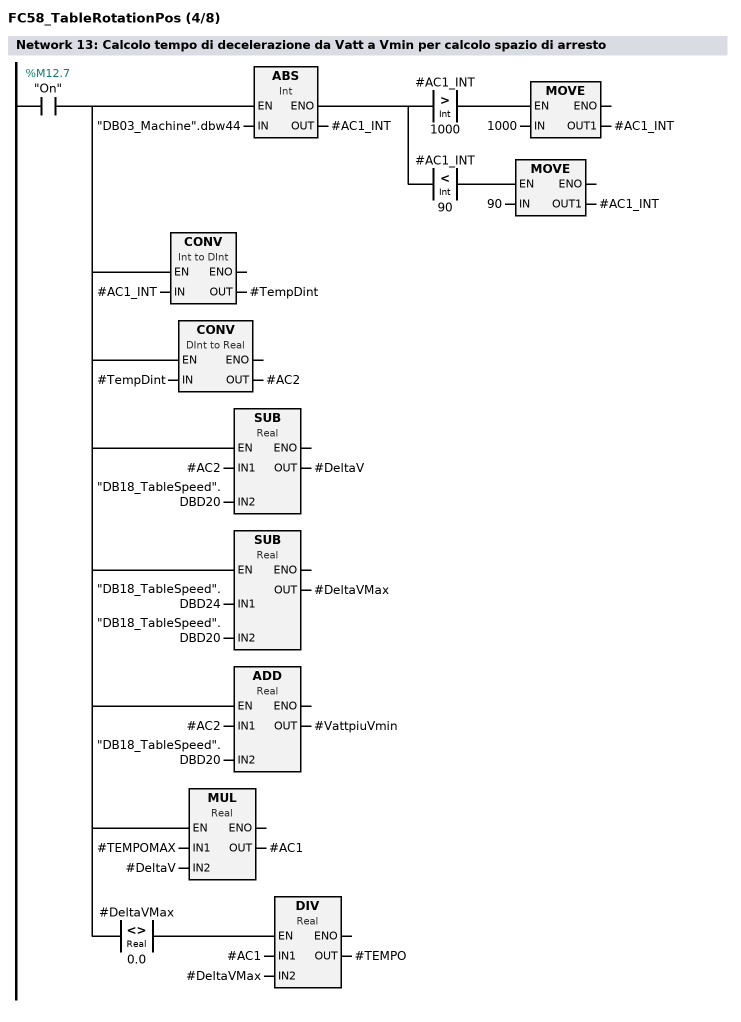
   RUNG wire#powerrail
      Contact( "On" )
      wire#w1
      { S7_Templates := "SrcType := Int" } Abs(in := "DB03_Machine".dbw44, out => #AC1_INT)
      wire#w2
      { S7_Templates := "SrcType := Int" } GT_Contact(in1 := #AC1_INT, in2 := 1000)
      Move(in := 1000, out1 => #AC1_INT)
   END_RUNG
   RUNG wire#w2
      { S7_Templates := "SrcType := Int" } LT_Contact(in1 := #AC1_INT, in2 := 90)
      Move(in := 90, out1 => #AC1_INT)
   END_RUNG
   RUNG wire#w1
      { S7_Templates := "[SrcType := Int, DestType := DInt]"; S7_GenerateENO := "TRUE" } Convert(in := #AC1_INT, out => #TempDint)
   END_RUNG
   RUNG wire#w1
      { S7_Templates := "[SrcType := DInt, DestType := Real]"; S7_GenerateENO := "TRUE" } Convert(in := #TempDint, out => #AC2)
   END_RUNG
   RUNG wire#w1
      { S7_Templates := "SrcType := Real"; S7_GenerateENO := "TRUE" } Sub(in1 := #AC2, in2 := "DB18_TableSpeed".DBD20, out => #DeltaV)
   END_RUNG
   RUNG wire#w1
      { S7_Templates := "SrcType := Real"; S7_GenerateENO := "TRUE" } Sub(in1 := "DB18_TableSpeed".DBD24, in2 := "DB18_TableSpeed".DBD20, out => #DeltaVMax)
   END_RUNG
   RUNG wire#w1
      { S7_Templates := "SrcType := Real"; S7_GenerateENO := "TRUE" } Add(in1 := #AC2, in2 := "DB18_TableSpeed".DBD20, out => #VattpiuVmin)
   END_RUNG
   RUNG wire#w1
      { S7_Templates := "SrcType := Real"; S7_GenerateENO := "TRUE" } Mul(in1 := #TEMPOMAX, in2 := #DeltaV, out => #AC1)
   END_RUNG
   RUNG wire#w1
      { S7_Templates := "SrcType := Real" } NE_Contact(in1 := #DeltaVMax, in2 := 0.0)
      { S7_Templates := "SrcType := Real"; S7_GenerateENO := "TRUE" } Div(in1 := #AC1, in2 := #DeltaVMax, out => #TEMPO)
   END_RUNG
   // the same network as SCL:
   IF "On" THEN #AC1_INT := ABS("DB03_Machine".dbw44); END_IF;
   IF "On" AND (#AC1_INT > 1000) THEN #AC1_INT := 1000; END_IF;
   IF "On" AND (#AC1_INT < 90) THEN #AC1_INT := 90; END_IF;
   IF "On" THEN
       #TempDint := INT_TO_DINT(#AC1_INT);
       #AC2 := DINT_TO_REAL(#TempDint);
       #DeltaV := #AC2 - "DB18_TableSpeed".DBD20;
       #DeltaVMax := "DB18_TableSpeed".DBD24 - "DB18_TableSpeed".DBD20;
       #VattpiuVmin := #AC2 + "DB18_TableSpeed".DBD20;
       #AC1 := #TEMPOMAX * #DeltaV;
   END_IF;
   IF "On" AND (#DeltaVMax <> 0.0) THEN #TEMPO := #AC1 / #DeltaVMax; END_IF;
END_REGION

REGION Network 14: Decelerazione
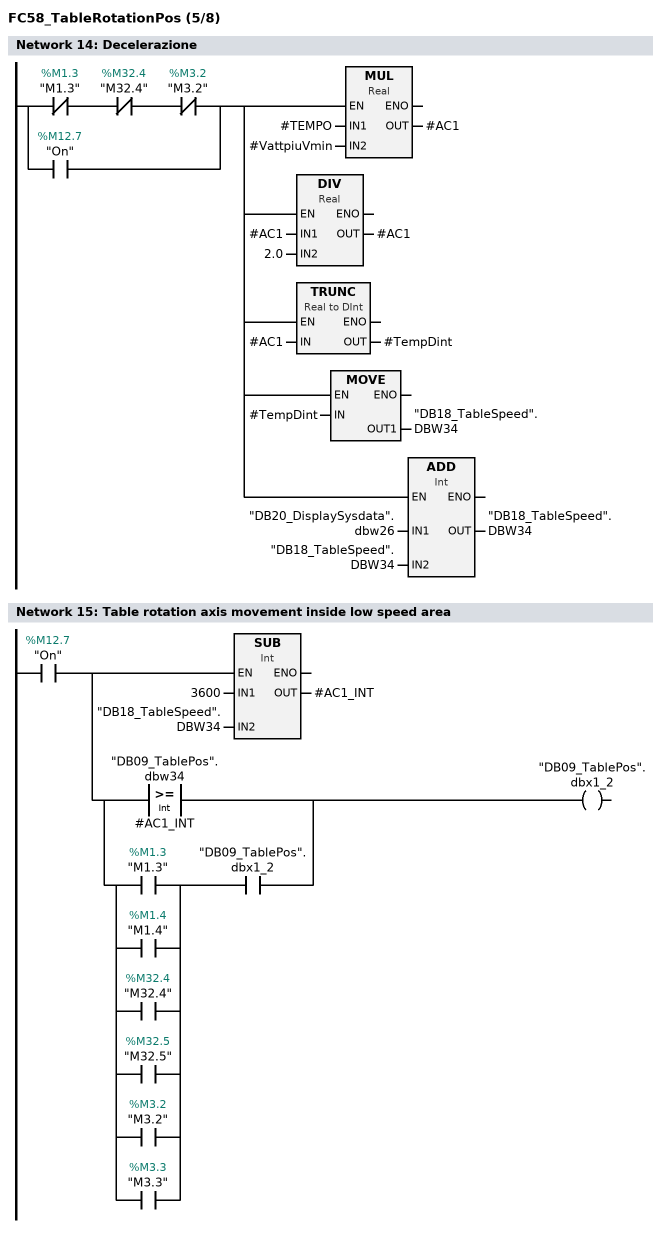
   RUNG wire#powerrail
      I_Contact( "M1.3" )
      I_Contact( "M32.4" )
      I_Contact( "M3.2" )
      wire#w1
      { S7_Templates := "SrcType := Real"; S7_GenerateENO := "TRUE" } Mul(in1 := #TEMPO, in2 := #VattpiuVmin, out => #AC1)
   END_RUNG
   RUNG wire#powerrail
      Contact( "On" )
   END_RUNG wire#w1
   RUNG wire#w1
      { S7_Templates := "SrcType := Real"; S7_GenerateENO := "TRUE" } Div(in1 := #AC1, in2 := 2.0, out => #AC1)
   END_RUNG
   RUNG wire#w1
      { S7_Templates := "[SrcType := Real, DestType := DInt]"; S7_GenerateENO := "TRUE" } Trunc(in := #AC1, out => #TempDint)
   END_RUNG
   RUNG wire#w1
      { S7_GenerateENO := "TRUE" } Move(in := #TempDint, out1 => "DB18_TableSpeed".DBW34)
   END_RUNG
   RUNG wire#w1
      { S7_Templates := "SrcType := Int"; S7_GenerateENO := "TRUE" } Add(in1 := "DB20_DisplaySysdata".dbw26, in2 := "DB18_TableSpeed".DBW34, out => "DB18_TableSpeed".DBW34)
   END_RUNG
   // the same network as SCL:
   IF (NOT "M1.3" AND NOT "M32.4" AND NOT "M3.2") OR "On" THEN
       #AC1 := #TEMPO * #VattpiuVmin;
       #AC1 := #AC1 / 2.0;
       #TempDint := TRUNC(#AC1);
       "DB18_TableSpeed".DBW34 := #TempDint;
       "DB18_TableSpeed".DBW34 := "DB20_DisplaySysdata".dbw26 + "DB18_TableSpeed".DBW34;
   END_IF;
END_REGION

REGION Network 15: Table rotation axis movement inside low speed area
   RUNG wire#powerrail
      Contact( "On" )
      wire#w1
      { S7_Templates := "SrcType := Int"; S7_GenerateENO := "TRUE" } Sub(in1 := 3600, in2 := "DB18_TableSpeed".DBW34, out => #AC1_INT)
   END_RUNG
   RUNG wire#w1
      { S7_Templates := "SrcType := Int" } GE_Contact(in1 := "DB09_TablePos".dbw34, in2 := #AC1_INT)
      wire#w2
      Coil( "DB09_TablePos".dbx1_2 )
   END_RUNG
   RUNG wire#w1
      Contact( "M1.3" )
      wire#w3
      Contact( "DB09_TablePos".dbx1_2 )
   END_RUNG wire#w2
   RUNG wire#w1
      Contact( "M1.4" )
   END_RUNG wire#w3
   RUNG wire#w1
      Contact( "M32.4" )
   END_RUNG wire#w3
   RUNG wire#w1
      Contact( "M32.5" )
   END_RUNG wire#w3
   RUNG wire#w1
      Contact( "M3.2" )
   END_RUNG wire#w3
   RUNG wire#w1
      Contact( "M3.3" )
   END_RUNG wire#w3
   // the same network as SCL:
   IF "On" THEN #AC1_INT := 3600 - "DB18_TableSpeed".DBW34; END_IF;
   "DB09_TablePos".dbx1_2 := "On" AND (("DB09_TablePos".dbw34 >= #AC1_INT) OR (("M1.3" OR "M1.4" OR "M32.4" OR "M32.5" OR "M3.2" OR "M3.3") AND "DB09_TablePos".dbx1_2));
END_REGION

REGION Network 16: Table rotation position loading/Unloading
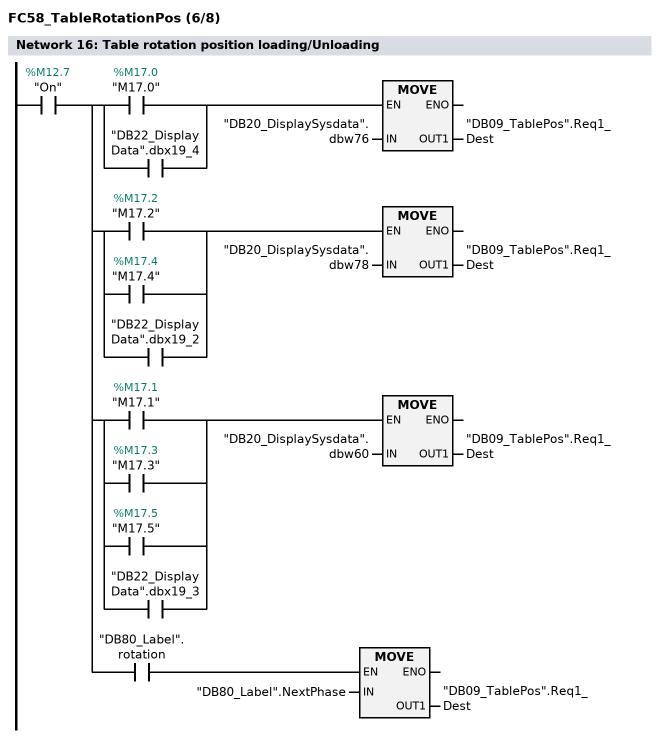
   RUNG wire#powerrail
      Contact( "On" )
      wire#w1
      Contact( "M17.0" )
      wire#w2
      { S7_GenerateENO := "TRUE" } Move(in := "DB20_DisplaySysdata".dbw76, out1 => "DB09_TablePos".Req1_Dest)
   END_RUNG
   RUNG wire#w1
      Contact( "DB22_DisplayData".dbx19_4 )
   END_RUNG wire#w2
   RUNG wire#w1
      Contact( "M17.2" )
      wire#w3
      { S7_GenerateENO := "TRUE" } Move(in := "DB20_DisplaySysdata".dbw78, out1 => "DB09_TablePos".Req1_Dest)
   END_RUNG
   RUNG wire#w1
      Contact( "M17.4" )
   END_RUNG wire#w3
   RUNG wire#w1
      Contact( "DB22_DisplayData".dbx19_2 )
   END_RUNG wire#w3
   RUNG wire#w1
      Contact( "M17.1" )
      wire#w4
      { S7_GenerateENO := "TRUE" } Move(in := "DB20_DisplaySysdata".dbw60, out1 => "DB09_TablePos".Req1_Dest)
   END_RUNG
   RUNG wire#w1
      Contact( "M17.3" )
   END_RUNG wire#w4
   RUNG wire#w1
      Contact( "M17.5" )
   END_RUNG wire#w4
   RUNG wire#w1
      Contact( "DB22_DisplayData".dbx19_3 )
   END_RUNG wire#w4
   RUNG wire#w1
      Contact( "DB80_Label".rotation )
      { S7_GenerateENO := "TRUE" } Move(in := "DB80_Label".NextPhase, out1 => "DB09_TablePos".Req1_Dest)
   END_RUNG
   // the same network as SCL:
   IF "On" AND ("M17.0" OR "DB22_DisplayData".dbx19_4) THEN
       "DB09_TablePos".Req1_Dest := "DB20_DisplaySysdata".dbw76;
   END_IF;
   IF "On" AND ("M17.2" OR "M17.4" OR "DB22_DisplayData".dbx19_2) THEN
       "DB09_TablePos".Req1_Dest := "DB20_DisplaySysdata".dbw78;
   END_IF;
   IF "On" AND ("M17.1" OR "M17.3" OR "M17.5" OR "DB22_DisplayData".dbx19_3) THEN
       "DB09_TablePos".Req1_Dest := "DB20_DisplaySysdata".dbw60;
   END_IF;
   IF "On" AND "DB80_Label".rotation THEN "DB09_TablePos".Req1_Dest := "DB80_Label".NextPhase; END_IF;
END_REGION

REGION Network 17
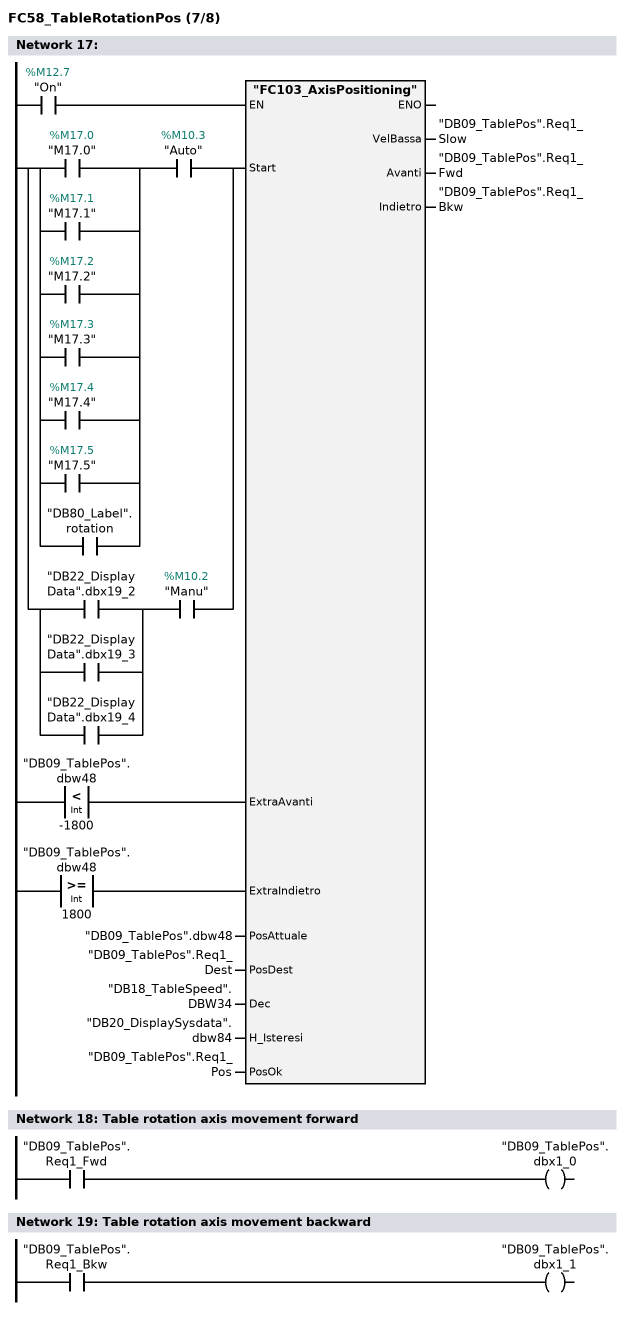
   RUNG wire#powerrail
      Contact( "On" )
      "FC103_AxisPositioning"(Start := wire#w3, ExtraAvanti := wire#w4, ExtraIndietro := wire#w5, PosAttuale := "DB09_TablePos".dbw48, PosDest := "DB09_TablePos".Req1_Dest, Dec := "DB18_TableSpeed".DBW34, H_Isteresi := "DB20_DisplaySysdata".dbw84, PosOk := "DB09_TablePos".Req1_Pos, VelBassa => "DB09_TablePos".Req1_Slow, Avanti => "DB09_TablePos".Req1_Fwd, Indietro => "DB09_TablePos".Req1_Bkw)
   END_RUNG
   RUNG wire#powerrail
      Contact( "M17.0" )
      wire#w1
      Contact( "Auto" )
   END_RUNG wire#w3
   RUNG wire#powerrail
      Contact( "M17.1" )
   END_RUNG wire#w1
   RUNG wire#powerrail
      Contact( "M17.2" )
   END_RUNG wire#w1
   RUNG wire#powerrail
      Contact( "M17.3" )
   END_RUNG wire#w1
   RUNG wire#powerrail
      Contact( "M17.4" )
   END_RUNG wire#w1
   RUNG wire#powerrail
      Contact( "M17.5" )
   END_RUNG wire#w1
   RUNG wire#powerrail
      Contact( "DB80_Label".rotation )
   END_RUNG wire#w1
   RUNG wire#powerrail
      Contact( "DB22_DisplayData".dbx19_2 )
      wire#w2
      Contact( "Manu" )
   END_RUNG wire#w3
   RUNG wire#powerrail
      Contact( "DB22_DisplayData".dbx19_3 )
   END_RUNG wire#w2
   RUNG wire#powerrail
      Contact( "DB22_DisplayData".dbx19_4 )
   END_RUNG wire#w2
   RUNG wire#powerrail
      { S7_Templates := "SrcType := Int" } LT_Contact(in1 := "DB09_TablePos".dbw48, in2 := -1800)
   END_RUNG wire#w4
   RUNG wire#powerrail
      { S7_Templates := "SrcType := Int" } GE_Contact(in1 := "DB09_TablePos".dbw48, in2 := 1800)
   END_RUNG wire#w5
   // the same network as SCL:
   IF "On" THEN
       "FC103_AxisPositioning"(Start := (("M17.0" OR "M17.1" OR "M17.2" OR "M17.3" OR "M17.4" OR "M17.5" OR "DB80_Label".rotation) AND "Auto") OR (("DB22_DisplayData".dbx19_2 OR "DB22_DisplayData".dbx19_3 OR "DB22_DisplayData".dbx19_4) AND "Manu"),
                               ExtraAvanti := "DB09_TablePos".dbw48 < (-1800),
                               ExtraIndietro := "DB09_TablePos".dbw48 >= 1800,
                               PosAttuale := "DB09_TablePos".dbw48,
                               PosDest := "DB09_TablePos".Req1_Dest,
                               Dec := "DB18_TableSpeed".DBW34,
                               H_Isteresi := "DB20_DisplaySysdata".dbw84,
                               PosOk := "DB09_TablePos".Req1_Pos,
                               VelBassa => "DB09_TablePos".Req1_Slow,
                               Avanti => "DB09_TablePos".Req1_Fwd,
                               Indietro => "DB09_TablePos".Req1_Bkw);
   END_IF;
END_REGION

REGION Network 18: Table rotation axis movement forward
   RUNG wire#powerrail
      Contact( "DB09_TablePos".Req1_Fwd )
      Coil( "DB09_TablePos".dbx1_0 )
   END_RUNG
   // the same network as SCL:
   "DB09_TablePos".dbx1_0 := "DB09_TablePos".Req1_Fwd;
END_REGION

REGION Network 19: Table rotation axis movement backward
   RUNG wire#powerrail
      Contact( "DB09_TablePos".Req1_Bkw )
      Coil( "DB09_TablePos".dbx1_1 )
   END_RUNG
   // the same network as SCL:
   "DB09_TablePos".dbx1_1 := "DB09_TablePos".Req1_Bkw;
END_REGION

REGION Network 20: Table rotation axis movement low speed
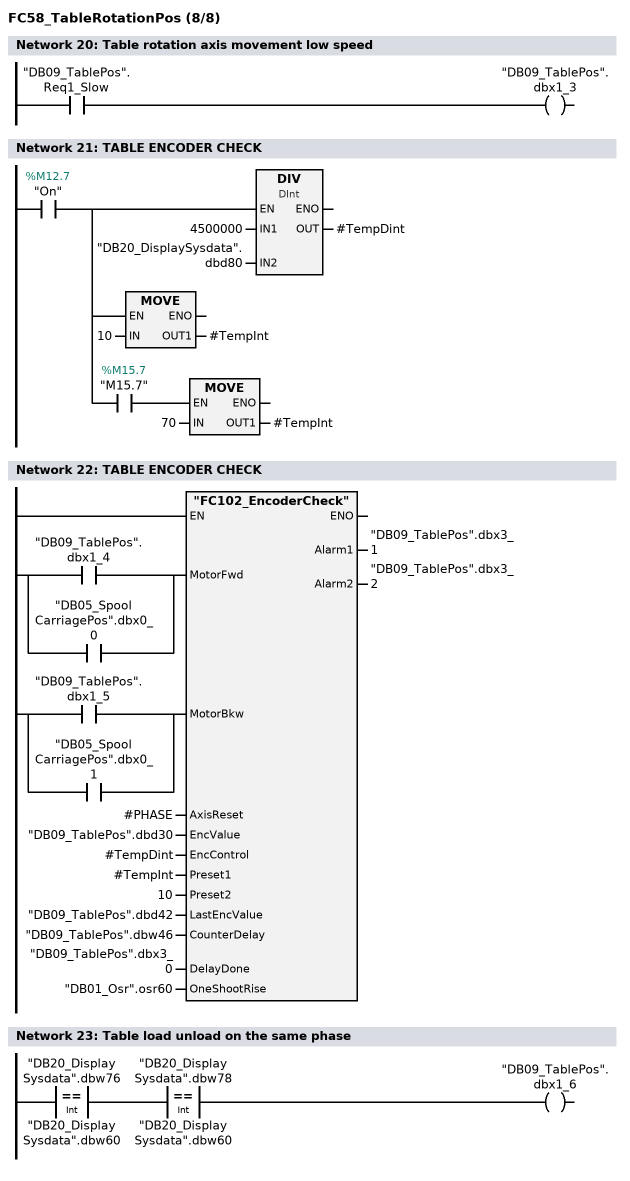
   RUNG wire#powerrail
      Contact( "DB09_TablePos".Req1_Slow )
      Coil( "DB09_TablePos".dbx1_3 )
   END_RUNG
   // the same network as SCL:
   "DB09_TablePos".dbx1_3 := "DB09_TablePos".Req1_Slow;
END_REGION

REGION Network 21: TABLE ENCODER CHECK
   RUNG wire#powerrail
      Contact( "On" )
      wire#w1
      { S7_Templates := "SrcType := DInt"; S7_GenerateENO := "TRUE" } Div(in1 := 4500000, in2 := "DB20_DisplaySysdata".dbd80, out => #TempDint)
   END_RUNG
   RUNG wire#w1
      { S7_GenerateENO := "TRUE" } Move(in := 10, out1 => #TempInt)
   END_RUNG
   RUNG wire#w1
      Contact( "M15.7" )
      { S7_GenerateENO := "TRUE" } Move(in := 70, out1 => #TempInt)
   END_RUNG
   // the same network as SCL:
   IF "On" THEN
       #TempDint := 4500000 / "DB20_DisplaySysdata".dbd80;
       #TempInt := 10;
   END_IF;
   IF "On" AND "M15.7" THEN #TempInt := 70; END_IF;
END_REGION

REGION Network 22: TABLE ENCODER CHECK
   RUNG wire#powerrail
      "FC102_EncoderCheck"(MotorFwd := wire#w1, MotorBkw := wire#w2, AxisReset := #PHASE, EncValue := "DB09_TablePos".dbd30, EncControl := #TempDint, Preset1 := #TempInt, Preset2 := 10, LastEncValue := "DB09_TablePos".dbd42, CounterDelay := "DB09_TablePos".dbw46, DelayDone := "DB09_TablePos".dbx3_0, OneShootRise := "DB01_Osr".osr60, Alarm1 => "DB09_TablePos".dbx3_1, Alarm2 => "DB09_TablePos".dbx3_2)
   END_RUNG
   RUNG wire#powerrail
      Contact( "DB09_TablePos".dbx1_4 )
   END_RUNG wire#w1
   RUNG wire#powerrail
      Contact( "DB05_SpoolCarriagePos".dbx0_0 )
   END_RUNG wire#w1
   RUNG wire#powerrail
      Contact( "DB09_TablePos".dbx1_5 )
   END_RUNG wire#w2
   RUNG wire#powerrail
      Contact( "DB05_SpoolCarriagePos".dbx0_1 )
   END_RUNG wire#w2
   // the same network as SCL:
   "FC102_EncoderCheck"(MotorFwd := "DB09_TablePos".dbx1_4 OR "DB05_SpoolCarriagePos".dbx0_0,
                        MotorBkw := "DB09_TablePos".dbx1_5 OR "DB05_SpoolCarriagePos".dbx0_1,
                        AxisReset := #PHASE,
                        EncValue := "DB09_TablePos".dbd30,
                        EncControl := #TempDint,
                        Preset1 := #TempInt,
                        Preset2 := 10,
                        LastEncValue := "DB09_TablePos".dbd42,
                        CounterDelay := "DB09_TablePos".dbw46,
                        DelayDone := "DB09_TablePos".dbx3_0,
                        OneShootRise := "DB01_Osr".osr60,
                        Alarm1 => "DB09_TablePos".dbx3_1,
                        Alarm2 => "DB09_TablePos".dbx3_2);
END_REGION

REGION Network 23: Table load unload on the same phase
   RUNG wire#powerrail
      { S7_Templates := "SrcType := Int" } EQ_Contact(in1 := "DB20_DisplaySysdata".dbw76, in2 := "DB20_DisplaySysdata".dbw60)
      { S7_Templates := "SrcType := Int" } EQ_Contact(in1 := "DB20_DisplaySysdata".dbw78, in2 := "DB20_DisplaySysdata".dbw60)
      Coil( "DB09_TablePos".dbx1_6 )
   END_RUNG
   // the same network as SCL:
   "DB09_TablePos".dbx1_6 := ("DB20_DisplaySysdata".dbw76 = "DB20_DisplaySysdata".dbw60) AND ("DB20_DisplaySysdata".dbw78 = "DB20_DisplaySysdata".dbw60);
END_REGION
END_FUNCTION

FUNCTION "FC06_TechnoplatCycle" : Void   // FC6, LAD
TITLE = Machine cycle
{ S7_Optimized_Access := 'FALSE' }
AUTHOR : Robopac
VERSION : 0.0
// stored: AutoNumber false, IsIECCheckEnabled false, SetENOAutomatically false, UDAEnableTagReadback false
   VAR_TEMP   // added for the SCL form of the ladder/FBD networks
      _w1 : Bool;
   END_VAR
BEGIN

REGION Network 1: Machine cycle: M0.0 Start cycle
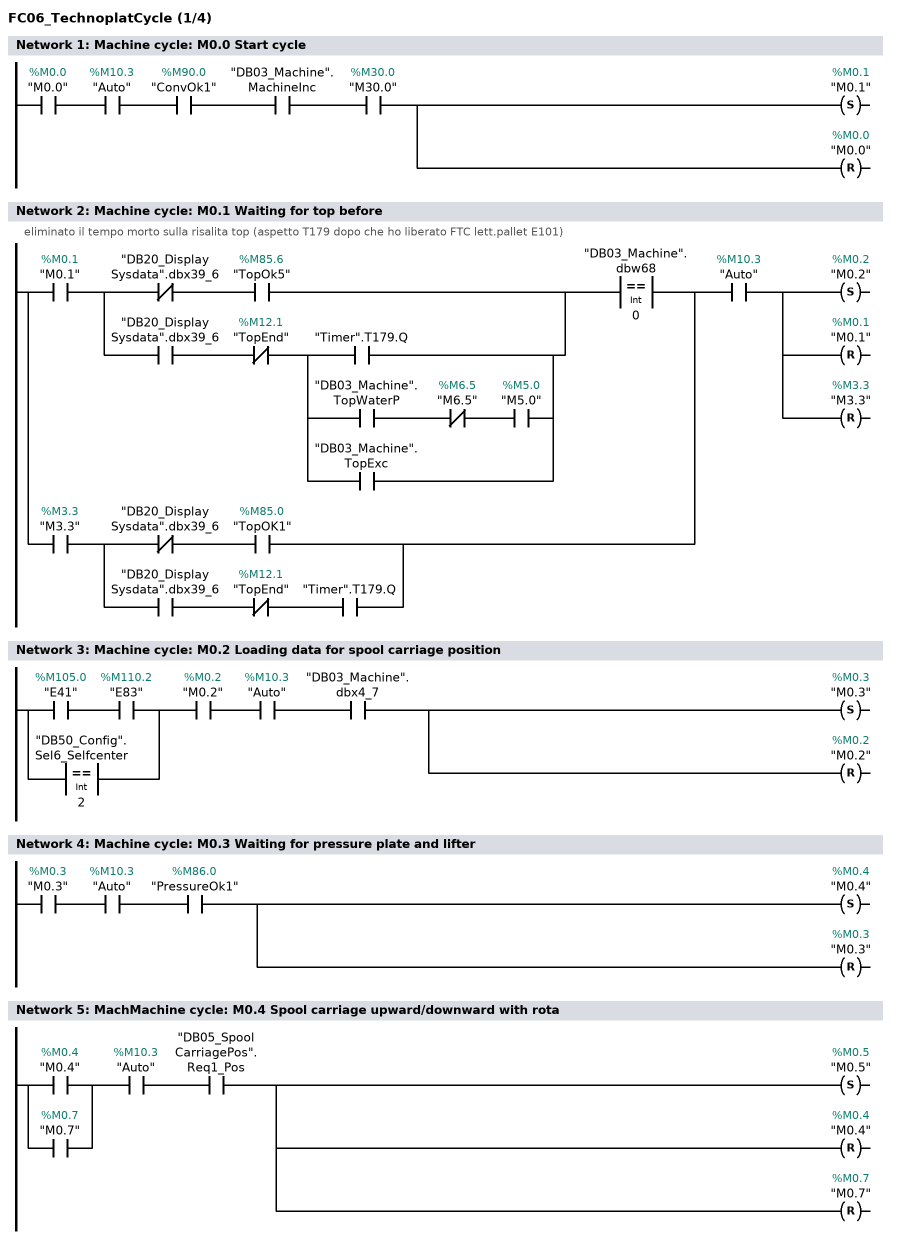
   RUNG wire#powerrail
      Contact( "M0.0" )
      Contact( "Auto" )
      Contact( "ConvOk1" )
      Contact( "DB03_Machine".MachineInc )
      Contact( "M30.0" )
      wire#w1
      S_Coil( "M0.1" )
   END_RUNG
   RUNG wire#w1
      R_Coil( "M0.0" )
   END_RUNG
   // the same network as SCL:
   IF "M0.0" AND "Auto" AND "ConvOk1" AND "DB03_Machine".MachineInc AND "M30.0" THEN
       "M0.1" := TRUE;
       "M0.0" := FALSE;
   END_IF;
END_REGION

REGION Network 2: Machine cycle: M0.1 Waiting for top before
   // eliminato il tempo morto sulla risalita top (aspetto T179 dopo che ho liberato FTC lett.pallet E101)
   RUNG wire#powerrail
      Contact( "M0.1" )
      wire#w1
      I_Contact( "DB20_DisplaySysdata".dbx39_6 )
      Contact( "TopOk5" )
      wire#w2
      { S7_Templates := "SrcType := Int" } EQ_Contact(in1 := "DB03_Machine".dbw68, in2 := 0)
      wire#w4
      Contact( "Auto" )
      wire#w6
      S_Coil( "M0.2" )
   END_RUNG
   RUNG wire#w1
      Contact( "DB20_DisplaySysdata".dbx39_6 )
      I_Contact( "TopEnd" )
      wire#w3
      Contact( "Timer".T179.Q )
   END_RUNG wire#w2
   RUNG wire#w3
      Contact( "DB03_Machine".TopWaterP )
      I_Contact( "M6.5" )
      Contact( "M5.0" )
   END_RUNG wire#w2
   RUNG wire#w3
      Contact( "DB03_Machine".TopExc )
   END_RUNG wire#w2
   RUNG wire#powerrail
      Contact( "M3.3" )
      wire#w5
      I_Contact( "DB20_DisplaySysdata".dbx39_6 )
      Contact( "TopOK1" )
   END_RUNG wire#w4
   RUNG wire#w5
      Contact( "DB20_DisplaySysdata".dbx39_6 )
      I_Contact( "TopEnd" )
      Contact( "Timer".T179.Q )
   END_RUNG wire#w4
   RUNG wire#w6
      R_Coil( "M0.1" )
   END_RUNG
   RUNG wire#w6
      R_Coil( "M3.3" )
   END_RUNG
   // the same network as SCL:
   IF (("M0.1" AND ((NOT "DB20_DisplaySysdata".dbx39_6 AND "TopOk5") OR ("DB20_DisplaySysdata".dbx39_6 AND NOT "TopEnd" AND ("Timer".T179.Q OR ("DB03_Machine".TopWaterP AND NOT "M6.5" AND "M5.0") OR "DB03_Machine".TopExc))) AND ("DB03_Machine".dbw68 = 0)) OR ("M3.3" AND ((NOT "DB20_DisplaySysdata".dbx39_6 AND "TopOK1") OR ("DB20_DisplaySysdata".dbx39_6 AND NOT "TopEnd" AND "Timer".T179.Q)))) AND "Auto" THEN
       "M0.2" := TRUE;
   END_IF;
   #_w1 := (("M0.1" AND ((NOT "DB20_DisplaySysdata".dbx39_6 AND "TopOk5") OR ("DB20_DisplaySysdata".dbx39_6 AND NOT "TopEnd" AND ("Timer".T179.Q OR ("DB03_Machine".TopWaterP AND NOT "M6.5" AND "M5.0") OR "DB03_Machine".TopExc))) AND ("DB03_Machine".dbw68 = 0)) OR ("M3.3" AND ((NOT "DB20_DisplaySysdata".dbx39_6 AND "TopOK1") OR ("DB20_DisplaySysdata".dbx39_6 AND NOT "TopEnd" AND "Timer".T179.Q)))) AND "Auto";
   IF #_w1 THEN
       "M0.1" := FALSE;
       "M3.3" := FALSE;
   END_IF;
END_REGION

REGION Network 3: Machine cycle: M0.2 Loading data for spool carriage position
   RUNG wire#powerrail
      Contact( "E41" )
      Contact( "E83" )
      wire#w1
      Contact( "M0.2" )
      Contact( "Auto" )
      Contact( "DB03_Machine".dbx4_7 )
      wire#w2
      S_Coil( "M0.3" )
   END_RUNG
   RUNG wire#powerrail
      { S7_Templates := "SrcType := Int" } EQ_Contact(in1 := "DB50_Config".Sel6_Selfcenter, in2 := 2)
   END_RUNG wire#w1
   RUNG wire#w2
      R_Coil( "M0.2" )
   END_RUNG
   // the same network as SCL:
   IF (("E41" AND "E83") OR ("DB50_Config".Sel6_Selfcenter = 2)) AND "M0.2" AND "Auto" AND "DB03_Machine".dbx4_7 THEN
       "M0.3" := TRUE;
       "M0.2" := FALSE;
   END_IF;
END_REGION

REGION Network 4: Machine cycle: M0.3 Waiting for pressure plate and lifter
   RUNG wire#powerrail
      Contact( "M0.3" )
      Contact( "Auto" )
      Contact( "PressureOk1" )
      wire#w1
      S_Coil( "M0.4" )
   END_RUNG
   RUNG wire#w1
      R_Coil( "M0.3" )
   END_RUNG
   // the same network as SCL:
   IF "M0.3" AND "Auto" AND "PressureOk1" THEN
       "M0.4" := TRUE;
       "M0.3" := FALSE;
   END_IF;
END_REGION

REGION Network 5: MachMachine cycle: M0.4 Spool carriage upward/downward with rota
   RUNG wire#powerrail
      Contact( "M0.4" )
      wire#w1
      Contact( "Auto" )
      Contact( "DB05_SpoolCarriagePos".Req1_Pos )
      wire#w2
      S_Coil( "M0.5" )
   END_RUNG
   RUNG wire#powerrail
      Contact( "M0.7" )
   END_RUNG wire#w1
   RUNG wire#w2
      R_Coil( "M0.4" )
   END_RUNG
   RUNG wire#w2
      R_Coil( "M0.7" )
   END_RUNG
   // the same network as SCL:
   IF ("M0.4" OR "M0.7") AND "Auto" AND "DB05_SpoolCarriagePos".Req1_Pos THEN "M0.5" := TRUE; END_IF;
   #_w1 := ("M0.4" OR "M0.7") AND "Auto" AND "DB05_SpoolCarriagePos".Req1_Pos;
   IF #_w1 THEN
       "M0.4" := FALSE;
       "M0.7" := FALSE;
   END_IF;
END_REGION

REGION Network 6: Machine cycle: M0.5 Arm rotation - Arm revolution counter
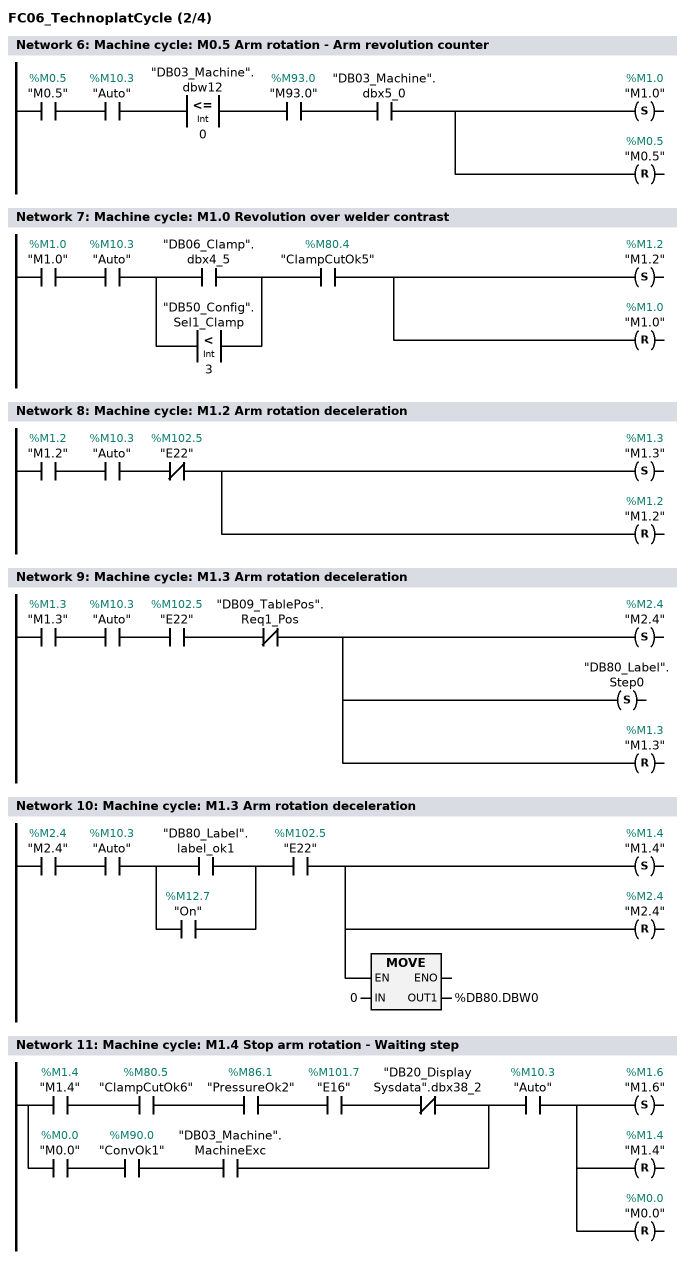
   RUNG wire#powerrail
      Contact( "M0.5" )
      Contact( "Auto" )
      { S7_Templates := "SrcType := Int" } LE_Contact(in1 := "DB03_Machine".dbw12, in2 := 0)
      Contact( "M93.0" )
      Contact( "DB03_Machine".dbx5_0 )
      wire#w1
      S_Coil( "M1.0" )
   END_RUNG
   RUNG wire#w1
      R_Coil( "M0.5" )
   END_RUNG
   // the same network as SCL:
   IF "M0.5" AND "Auto" AND ("DB03_Machine".dbw12 <= 0) AND "M93.0" AND "DB03_Machine".dbx5_0 THEN
       "M1.0" := TRUE;
       "M0.5" := FALSE;
   END_IF;
END_REGION

REGION Network 7: Machine cycle: M1.0 Revolution over welder contrast
   RUNG wire#powerrail
      Contact( "M1.0" )
      Contact( "Auto" )
      wire#w1
      Contact( "DB06_Clamp".dbx4_5 )
      wire#w2
      Contact( "ClampCutOk5" )
      wire#w3
      S_Coil( "M1.2" )
   END_RUNG
   RUNG wire#w1
      { S7_Templates := "SrcType := Int" } LT_Contact(in1 := "DB50_Config".Sel1_Clamp, in2 := 3)
   END_RUNG wire#w2
   RUNG wire#w3
      R_Coil( "M1.0" )
   END_RUNG
   // the same network as SCL:
   IF "M1.0" AND "Auto" AND ("DB06_Clamp".dbx4_5 OR ("DB50_Config".Sel1_Clamp < 3)) AND "ClampCutOk5" THEN
       "M1.2" := TRUE;
       "M1.0" := FALSE;
   END_IF;
END_REGION

REGION Network 8: Machine cycle: M1.2 Arm rotation deceleration
   RUNG wire#powerrail
      Contact( "M1.2" )
      Contact( "Auto" )
      I_Contact( "E22" )
      wire#w1
      S_Coil( "M1.3" )
   END_RUNG
   RUNG wire#w1
      R_Coil( "M1.2" )
   END_RUNG
   // the same network as SCL:
   IF "M1.2" AND "Auto" AND NOT "E22" THEN
       "M1.3" := TRUE;
       "M1.2" := FALSE;
   END_IF;
END_REGION

REGION Network 9: Machine cycle: M1.3 Arm rotation deceleration
   RUNG wire#powerrail
      Contact( "M1.3" )
      Contact( "Auto" )
      Contact( "E22" )
      I_Contact( "DB09_TablePos".Req1_Pos )
      wire#w1
      S_Coil( "M2.4" )
   END_RUNG
   RUNG wire#w1
      S_Coil( "DB80_Label".Step0 )
   END_RUNG
   RUNG wire#w1
      R_Coil( "M1.3" )
   END_RUNG
   // the same network as SCL:
   IF "M1.3" AND "Auto" AND "E22" AND NOT "DB09_TablePos".Req1_Pos THEN
       "M2.4" := TRUE;
       "DB80_Label".Step0 := TRUE;
       "M1.3" := FALSE;
   END_IF;
END_REGION

REGION Network 10: Machine cycle: M1.3 Arm rotation deceleration
   RUNG wire#powerrail
      Contact( "M2.4" )
      Contact( "Auto" )
      wire#w1
      Contact( "DB80_Label".label_ok1 )
      wire#w2
      Contact( "E22" )
      wire#w3
      S_Coil( "M1.4" )
   END_RUNG
   RUNG wire#w1
      Contact( "On" )
   END_RUNG wire#w2
   RUNG wire#w3
      R_Coil( "M2.4" )
   END_RUNG
   RUNG wire#w3
      { S7_GenerateENO := "TRUE" } Move(in := 0, out1 => %DB80.DBW0)
   END_RUNG
   // the same network as SCL:
   IF "M2.4" AND "Auto" AND ("DB80_Label".label_ok1 OR "On") AND "E22" THEN "M1.4" := TRUE; END_IF;
   #_w1 := "M2.4" AND "Auto" AND ("DB80_Label".label_ok1 OR "On") AND "E22";
   IF #_w1 THEN
       "M2.4" := FALSE;
       %DB80.DBW0 := 0;
   END_IF;
END_REGION

REGION Network 11: Machine cycle: M1.4 Stop arm rotation - Waiting step
   RUNG wire#powerrail
      Contact( "M1.4" )
      Contact( "ClampCutOk6" )
      Contact( "PressureOk2" )
      Contact( "E16" )
      I_Contact( "DB20_DisplaySysdata".dbx38_2 )
      wire#w1
      Contact( "Auto" )
      wire#w2
      S_Coil( "M1.6" )
   END_RUNG
   RUNG wire#powerrail
      Contact( "M0.0" )
      Contact( "ConvOk1" )
      Contact( "DB03_Machine".MachineExc )
   END_RUNG wire#w1
   RUNG wire#w2
      R_Coil( "M1.4" )
   END_RUNG
   RUNG wire#w2
      R_Coil( "M0.0" )
   END_RUNG
   // the same network as SCL:
   IF (("M1.4" AND "ClampCutOk6" AND "PressureOk2" AND "E16" AND NOT "DB20_DisplaySysdata".dbx38_2) OR ("M0.0" AND "ConvOk1" AND "DB03_Machine".MachineExc)) AND "Auto" THEN
       "M1.6" := TRUE;
   END_IF;
   #_w1 := (("M1.4" AND "ClampCutOk6" AND "PressureOk2" AND "E16" AND NOT "DB20_DisplaySysdata".dbx38_2) OR ("M0.0" AND "ConvOk1" AND "DB03_Machine".MachineExc)) AND "Auto";
   IF #_w1 THEN
       "M1.4" := FALSE;
       "M0.0" := FALSE;
   END_IF;
END_REGION

REGION Network 12: Machine cycle: M1.6 Pallet unload
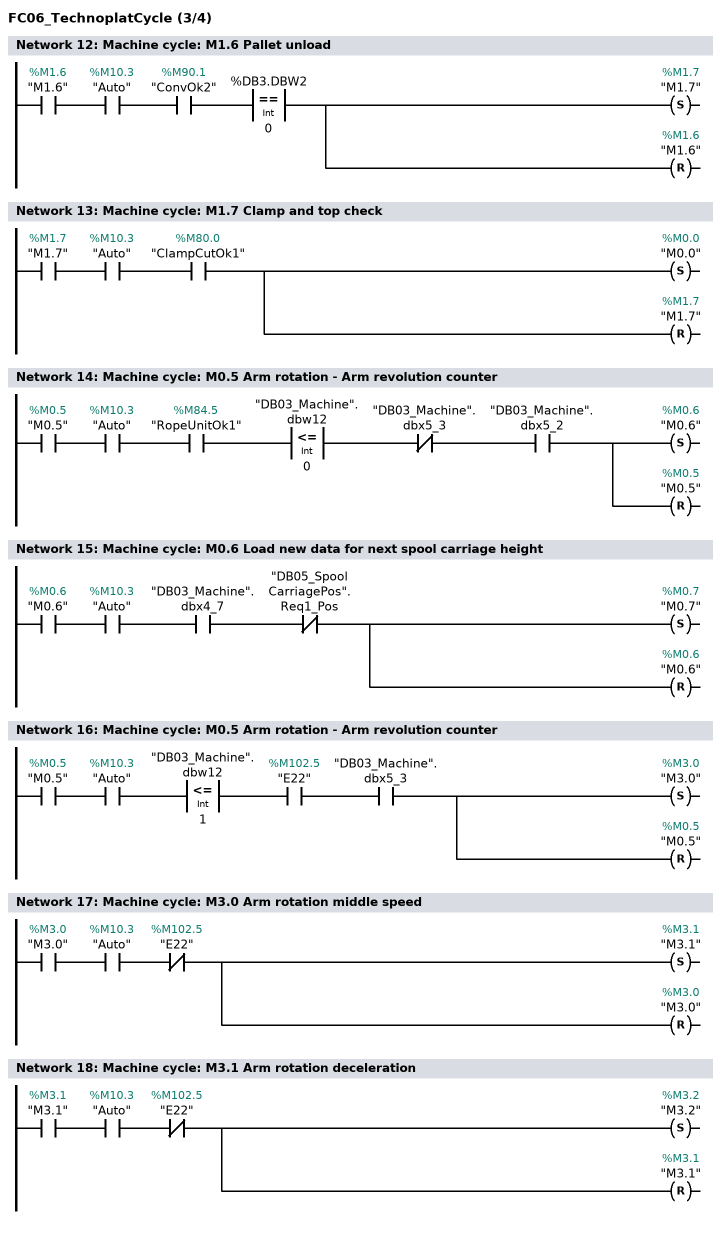
   RUNG wire#powerrail
      Contact( "M1.6" )
      Contact( "Auto" )
      Contact( "ConvOk2" )
      { S7_Templates := "SrcType := Int" } EQ_Contact(in1 := %DB3.DBW2, in2 := 0)
      wire#w1
      S_Coil( "M1.7" )
   END_RUNG
   RUNG wire#w1
      R_Coil( "M1.6" )
   END_RUNG
   // the same network as SCL:
   IF "M1.6" AND "Auto" AND "ConvOk2" AND (%DB3.DBW2 = 0) THEN
       "M1.7" := TRUE;
       "M1.6" := FALSE;
   END_IF;
END_REGION

REGION Network 13: Machine cycle: M1.7 Clamp and top check
   RUNG wire#powerrail
      Contact( "M1.7" )
      Contact( "Auto" )
      Contact( "ClampCutOk1" )
      wire#w1
      S_Coil( "M0.0" )
   END_RUNG
   RUNG wire#w1
      R_Coil( "M1.7" )
   END_RUNG
   // the same network as SCL:
   IF "M1.7" AND "Auto" AND "ClampCutOk1" THEN
       "M0.0" := TRUE;
       "M1.7" := FALSE;
   END_IF;
END_REGION

REGION Network 14: Machine cycle: M0.5 Arm rotation - Arm revolution counter
   RUNG wire#powerrail
      Contact( "M0.5" )
      Contact( "Auto" )
      Contact( "RopeUnitOk1" )
      { S7_Templates := "SrcType := Int" } LE_Contact(in1 := "DB03_Machine".dbw12, in2 := 0)
      I_Contact( "DB03_Machine".dbx5_3 )
      Contact( "DB03_Machine".dbx5_2 )
      wire#w1
      S_Coil( "M0.6" )
   END_RUNG
   RUNG wire#w1
      R_Coil( "M0.5" )
   END_RUNG
   // the same network as SCL:
   IF "M0.5" AND "Auto" AND "RopeUnitOk1" AND ("DB03_Machine".dbw12 <= 0) AND NOT "DB03_Machine".dbx5_3 AND "DB03_Machine".dbx5_2 THEN
       "M0.6" := TRUE;
       "M0.5" := FALSE;
   END_IF;
END_REGION

REGION Network 15: Machine cycle: M0.6 Load new data for next spool carriage height
   RUNG wire#powerrail
      Contact( "M0.6" )
      Contact( "Auto" )
      Contact( "DB03_Machine".dbx4_7 )
      I_Contact( "DB05_SpoolCarriagePos".Req1_Pos )
      wire#w1
      S_Coil( "M0.7" )
   END_RUNG
   RUNG wire#w1
      R_Coil( "M0.6" )
   END_RUNG
   // the same network as SCL:
   IF "M0.6" AND "Auto" AND "DB03_Machine".dbx4_7 AND NOT "DB05_SpoolCarriagePos".Req1_Pos THEN
       "M0.7" := TRUE;
       "M0.6" := FALSE;
   END_IF;
END_REGION

REGION Network 16: Machine cycle: M0.5 Arm rotation - Arm revolution counter
   RUNG wire#powerrail
      Contact( "M0.5" )
      Contact( "Auto" )
      { S7_Templates := "SrcType := Int" } LE_Contact(in1 := "DB03_Machine".dbw12, in2 := 1)
      Contact( "E22" )
      Contact( "DB03_Machine".dbx5_3 )
      wire#w1
      S_Coil( "M3.0" )
   END_RUNG
   RUNG wire#w1
      R_Coil( "M0.5" )
   END_RUNG
   // the same network as SCL:
   IF "M0.5" AND "Auto" AND ("DB03_Machine".dbw12 <= 1) AND "E22" AND "DB03_Machine".dbx5_3 THEN
       "M3.0" := TRUE;
       "M0.5" := FALSE;
   END_IF;
END_REGION

REGION Network 17: Machine cycle: M3.0 Arm rotation middle speed
   RUNG wire#powerrail
      Contact( "M3.0" )
      Contact( "Auto" )
      I_Contact( "E22" )
      wire#w1
      S_Coil( "M3.1" )
   END_RUNG
   RUNG wire#w1
      R_Coil( "M3.0" )
   END_RUNG
   // the same network as SCL:
   IF "M3.0" AND "Auto" AND NOT "E22" THEN
       "M3.1" := TRUE;
       "M3.0" := FALSE;
   END_IF;
END_REGION

REGION Network 18: Machine cycle: M3.1 Arm rotation deceleration
   RUNG wire#powerrail
      Contact( "M3.1" )
      Contact( "Auto" )
      I_Contact( "E22" )
      wire#w1
      S_Coil( "M3.2" )
   END_RUNG
   RUNG wire#w1
      R_Coil( "M3.1" )
   END_RUNG
   // the same network as SCL:
   IF "M3.1" AND "Auto" AND NOT "E22" THEN
       "M3.2" := TRUE;
       "M3.1" := FALSE;
   END_IF;
END_REGION

REGION Network 19: Machine cycle: M3.2 Arm rotation deceleration
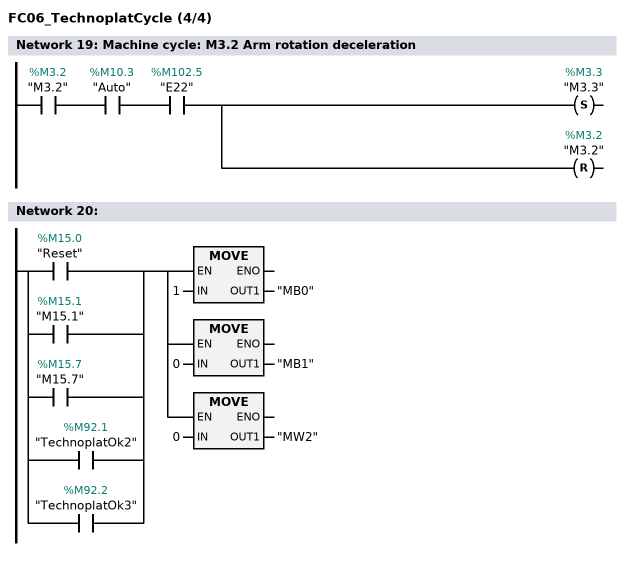
   RUNG wire#powerrail
      Contact( "M3.2" )
      Contact( "Auto" )
      Contact( "E22" )
      wire#w1
      S_Coil( "M3.3" )
   END_RUNG
   RUNG wire#w1
      R_Coil( "M3.2" )
   END_RUNG
   // the same network as SCL:
   IF "M3.2" AND "Auto" AND "E22" THEN
       "M3.3" := TRUE;
       "M3.2" := FALSE;
   END_IF;
END_REGION

REGION Network 20
   RUNG wire#powerrail
      Contact( "Reset" )
      wire#w1
      { S7_GenerateENO := "TRUE" } Move(in := 1, out1 => "MB0")
   END_RUNG
   RUNG wire#powerrail
      Contact( "M15.1" )
   END_RUNG wire#w1
   RUNG wire#powerrail
      Contact( "M15.7" )
   END_RUNG wire#w1
   RUNG wire#powerrail
      Contact( "TechnoplatOk2" )
   END_RUNG wire#w1
   RUNG wire#powerrail
      Contact( "TechnoplatOk3" )
   END_RUNG wire#w1
   RUNG wire#w1
      { S7_GenerateENO := "TRUE" } Move(in := 0, out1 => "MB1")
   END_RUNG
   RUNG wire#w1
      { S7_GenerateENO := "TRUE" } Move(in := 0, out1 => "MW2")
   END_RUNG
   // the same network as SCL:
   IF "Reset" OR "M15.1" OR "M15.7" OR "TechnoplatOk2" OR "TechnoplatOk3" THEN
       "MB0" := 1;
       "MB1" := 0;
       "MW2" := 0;
   END_IF;
END_REGION
END_FUNCTION

FUNCTION "FC80_Label" : Void   // FC80, LAD
TITLE = Label device
{ S7_Optimized_Access := 'FALSE' }
VERSION : 0.1
// stored: AutoNumber false, IsIECCheckEnabled false, SetENOAutomatically false, UDAEnableTagReadback false
BEGIN

REGION Network 1: Label arm in home position for pallet transit
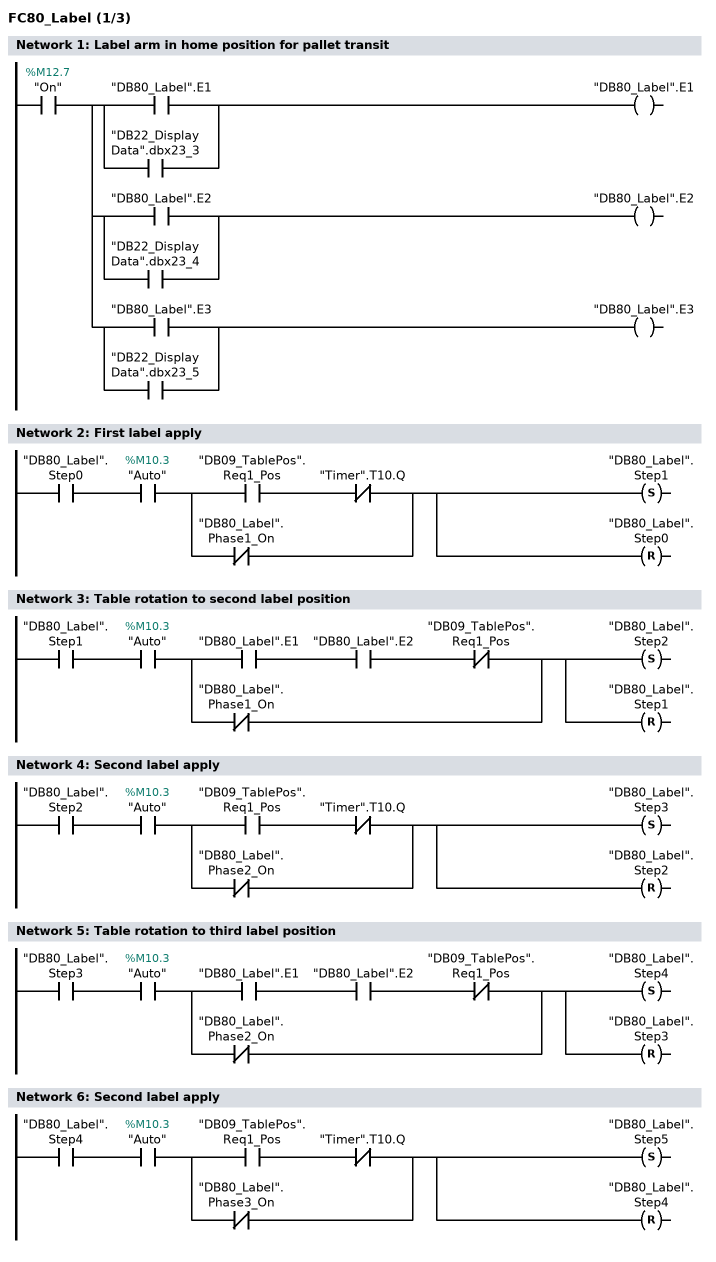
   RUNG wire#powerrail
      Contact( "On" )
      wire#w1
      Contact( "DB80_Label".E1 )
      wire#w2
      Coil( "DB80_Label".E1 )
   END_RUNG
   RUNG wire#w1
      Contact( "DB22_DisplayData".dbx23_3 )
   END_RUNG wire#w2
   RUNG wire#w1
      Contact( "DB80_Label".E2 )
      wire#w3
      Coil( "DB80_Label".E2 )
   END_RUNG
   RUNG wire#w1
      Contact( "DB22_DisplayData".dbx23_4 )
   END_RUNG wire#w3
   RUNG wire#w1
      Contact( "DB80_Label".E3 )
      wire#w4
      Coil( "DB80_Label".E3 )
   END_RUNG
   RUNG wire#w1
      Contact( "DB22_DisplayData".dbx23_5 )
   END_RUNG wire#w4
   // the same network as SCL:
   "DB80_Label".E1 := "On" AND ("DB80_Label".E1 OR "DB22_DisplayData".dbx23_3);
   "DB80_Label".E2 := "On" AND ("DB80_Label".E2 OR "DB22_DisplayData".dbx23_4);
   "DB80_Label".E3 := "On" AND ("DB80_Label".E3 OR "DB22_DisplayData".dbx23_5);
END_REGION

REGION Network 2: First label apply
   RUNG wire#powerrail
      Contact( "DB80_Label".Step0 )
      Contact( "Auto" )
      wire#w1
      Contact( "DB09_TablePos".Req1_Pos )
      I_Contact( "Timer".T10.Q )
      wire#w2
      S_Coil( "DB80_Label".Step1 )
   END_RUNG
   RUNG wire#w1
      I_Contact( "DB80_Label".Phase1_On )
   END_RUNG wire#w2
   RUNG wire#w2
      R_Coil( "DB80_Label".Step0 )
   END_RUNG
   // the same network as SCL:
   IF "DB80_Label".Step0 AND "Auto" AND (("DB09_TablePos".Req1_Pos AND NOT "Timer".T10.Q) OR NOT "DB80_Label".Phase1_On) THEN
       "DB80_Label".Step1 := TRUE;
       "DB80_Label".Step0 := FALSE;
   END_IF;
END_REGION

REGION Network 3: Table rotation to second label position
   RUNG wire#powerrail
      Contact( "DB80_Label".Step1 )
      Contact( "Auto" )
      wire#w1
      Contact( "DB80_Label".E1 )
      Contact( "DB80_Label".E2 )
      I_Contact( "DB09_TablePos".Req1_Pos )
      wire#w2
      S_Coil( "DB80_Label".Step2 )
   END_RUNG
   RUNG wire#w1
      I_Contact( "DB80_Label".Phase1_On )
   END_RUNG wire#w2
   RUNG wire#w2
      R_Coil( "DB80_Label".Step1 )
   END_RUNG
   // the same network as SCL:
   IF "DB80_Label".Step1 AND "Auto" AND (("DB80_Label".E1 AND "DB80_Label".E2 AND NOT "DB09_TablePos".Req1_Pos) OR NOT "DB80_Label".Phase1_On) THEN
       "DB80_Label".Step2 := TRUE;
       "DB80_Label".Step1 := FALSE;
   END_IF;
END_REGION

REGION Network 4: Second label apply
   RUNG wire#powerrail
      Contact( "DB80_Label".Step2 )
      Contact( "Auto" )
      wire#w1
      Contact( "DB09_TablePos".Req1_Pos )
      I_Contact( "Timer".T10.Q )
      wire#w2
      S_Coil( "DB80_Label".Step3 )
   END_RUNG
   RUNG wire#w1
      I_Contact( "DB80_Label".Phase2_On )
   END_RUNG wire#w2
   RUNG wire#w2
      R_Coil( "DB80_Label".Step2 )
   END_RUNG
   // the same network as SCL:
   IF "DB80_Label".Step2 AND "Auto" AND (("DB09_TablePos".Req1_Pos AND NOT "Timer".T10.Q) OR NOT "DB80_Label".Phase2_On) THEN
       "DB80_Label".Step3 := TRUE;
       "DB80_Label".Step2 := FALSE;
   END_IF;
END_REGION

REGION Network 5: Table rotation to third label position
   RUNG wire#powerrail
      Contact( "DB80_Label".Step3 )
      Contact( "Auto" )
      wire#w1
      Contact( "DB80_Label".E1 )
      Contact( "DB80_Label".E2 )
      I_Contact( "DB09_TablePos".Req1_Pos )
      wire#w2
      S_Coil( "DB80_Label".Step4 )
   END_RUNG
   RUNG wire#w1
      I_Contact( "DB80_Label".Phase2_On )
   END_RUNG wire#w2
   RUNG wire#w2
      R_Coil( "DB80_Label".Step3 )
   END_RUNG
   // the same network as SCL:
   IF "DB80_Label".Step3 AND "Auto" AND (("DB80_Label".E1 AND "DB80_Label".E2 AND NOT "DB09_TablePos".Req1_Pos) OR NOT "DB80_Label".Phase2_On) THEN
       "DB80_Label".Step4 := TRUE;
       "DB80_Label".Step3 := FALSE;
   END_IF;
END_REGION

REGION Network 6: Second label apply
   RUNG wire#powerrail
      Contact( "DB80_Label".Step4 )
      Contact( "Auto" )
      wire#w1
      Contact( "DB09_TablePos".Req1_Pos )
      I_Contact( "Timer".T10.Q )
      wire#w2
      S_Coil( "DB80_Label".Step5 )
   END_RUNG
   RUNG wire#w1
      I_Contact( "DB80_Label".Phase3_On )
   END_RUNG wire#w2
   RUNG wire#w2
      R_Coil( "DB80_Label".Step4 )
   END_RUNG
   // the same network as SCL:
   IF "DB80_Label".Step4 AND "Auto" AND (("DB09_TablePos".Req1_Pos AND NOT "Timer".T10.Q) OR NOT "DB80_Label".Phase3_On) THEN
       "DB80_Label".Step5 := TRUE;
       "DB80_Label".Step4 := FALSE;
   END_IF;
END_REGION

REGION Network 7: Table rotation to fourth label position
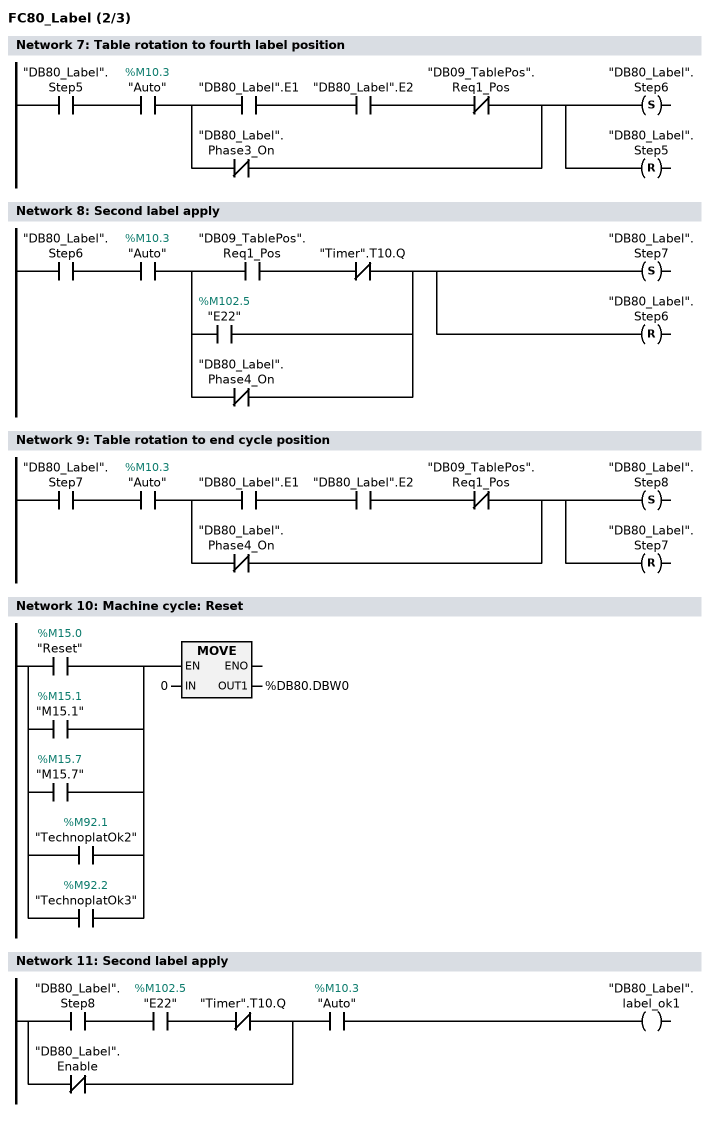
   RUNG wire#powerrail
      Contact( "DB80_Label".Step5 )
      Contact( "Auto" )
      wire#w1
      Contact( "DB80_Label".E1 )
      Contact( "DB80_Label".E2 )
      I_Contact( "DB09_TablePos".Req1_Pos )
      wire#w2
      S_Coil( "DB80_Label".Step6 )
   END_RUNG
   RUNG wire#w1
      I_Contact( "DB80_Label".Phase3_On )
   END_RUNG wire#w2
   RUNG wire#w2
      R_Coil( "DB80_Label".Step5 )
   END_RUNG
   // the same network as SCL:
   IF "DB80_Label".Step5 AND "Auto" AND (("DB80_Label".E1 AND "DB80_Label".E2 AND NOT "DB09_TablePos".Req1_Pos) OR NOT "DB80_Label".Phase3_On) THEN
       "DB80_Label".Step6 := TRUE;
       "DB80_Label".Step5 := FALSE;
   END_IF;
END_REGION

REGION Network 8: Second label apply
   RUNG wire#powerrail
      Contact( "DB80_Label".Step6 )
      Contact( "Auto" )
      wire#w1
      Contact( "DB09_TablePos".Req1_Pos )
      I_Contact( "Timer".T10.Q )
      wire#w2
      S_Coil( "DB80_Label".Step7 )
   END_RUNG
   RUNG wire#w1
      Contact( "E22" )
   END_RUNG wire#w2
   RUNG wire#w1
      I_Contact( "DB80_Label".Phase4_On )
   END_RUNG wire#w2
   RUNG wire#w2
      R_Coil( "DB80_Label".Step6 )
   END_RUNG
   // the same network as SCL:
   IF "DB80_Label".Step6 AND "Auto" AND (("DB09_TablePos".Req1_Pos AND NOT "Timer".T10.Q) OR "E22" OR NOT "DB80_Label".Phase4_On) THEN
       "DB80_Label".Step7 := TRUE;
       "DB80_Label".Step6 := FALSE;
   END_IF;
END_REGION

REGION Network 9: Table rotation to end cycle position
   RUNG wire#powerrail
      Contact( "DB80_Label".Step7 )
      Contact( "Auto" )
      wire#w1
      Contact( "DB80_Label".E1 )
      Contact( "DB80_Label".E2 )
      I_Contact( "DB09_TablePos".Req1_Pos )
      wire#w2
      S_Coil( "DB80_Label".Step8 )
   END_RUNG
   RUNG wire#w1
      I_Contact( "DB80_Label".Phase4_On )
   END_RUNG wire#w2
   RUNG wire#w2
      R_Coil( "DB80_Label".Step7 )
   END_RUNG
   // the same network as SCL:
   IF "DB80_Label".Step7 AND "Auto" AND (("DB80_Label".E1 AND "DB80_Label".E2 AND NOT "DB09_TablePos".Req1_Pos) OR NOT "DB80_Label".Phase4_On) THEN
       "DB80_Label".Step8 := TRUE;
       "DB80_Label".Step7 := FALSE;
   END_IF;
END_REGION

REGION Network 10: Machine cycle: Reset
   RUNG wire#powerrail
      Contact( "Reset" )
      wire#w1
      { S7_GenerateENO := "TRUE" } Move(in := 0, out1 => %DB80.DBW0)
   END_RUNG
   RUNG wire#powerrail
      Contact( "M15.1" )
   END_RUNG wire#w1
   RUNG wire#powerrail
      Contact( "M15.7" )
   END_RUNG wire#w1
   RUNG wire#powerrail
      Contact( "TechnoplatOk2" )
   END_RUNG wire#w1
   RUNG wire#powerrail
      Contact( "TechnoplatOk3" )
   END_RUNG wire#w1
   // the same network as SCL:
   IF "Reset" OR "M15.1" OR "M15.7" OR "TechnoplatOk2" OR "TechnoplatOk3" THEN %DB80.DBW0 := 0; END_IF;
END_REGION

REGION Network 11: Second label apply
   RUNG wire#powerrail
      Contact( "DB80_Label".Step8 )
      Contact( "E22" )
      I_Contact( "Timer".T10.Q )
      wire#w1
      Contact( "Auto" )
      Coil( "DB80_Label".label_ok1 )
   END_RUNG
   RUNG wire#powerrail
      I_Contact( "DB80_Label".Enable )
   END_RUNG wire#w1
   // the same network as SCL:
   "DB80_Label".label_ok1 := (("DB80_Label".Step8 AND "E22" AND NOT "Timer".T10.Q) OR NOT "DB80_Label".Enable) AND "Auto";
END_REGION

REGION Network 12: Label phases
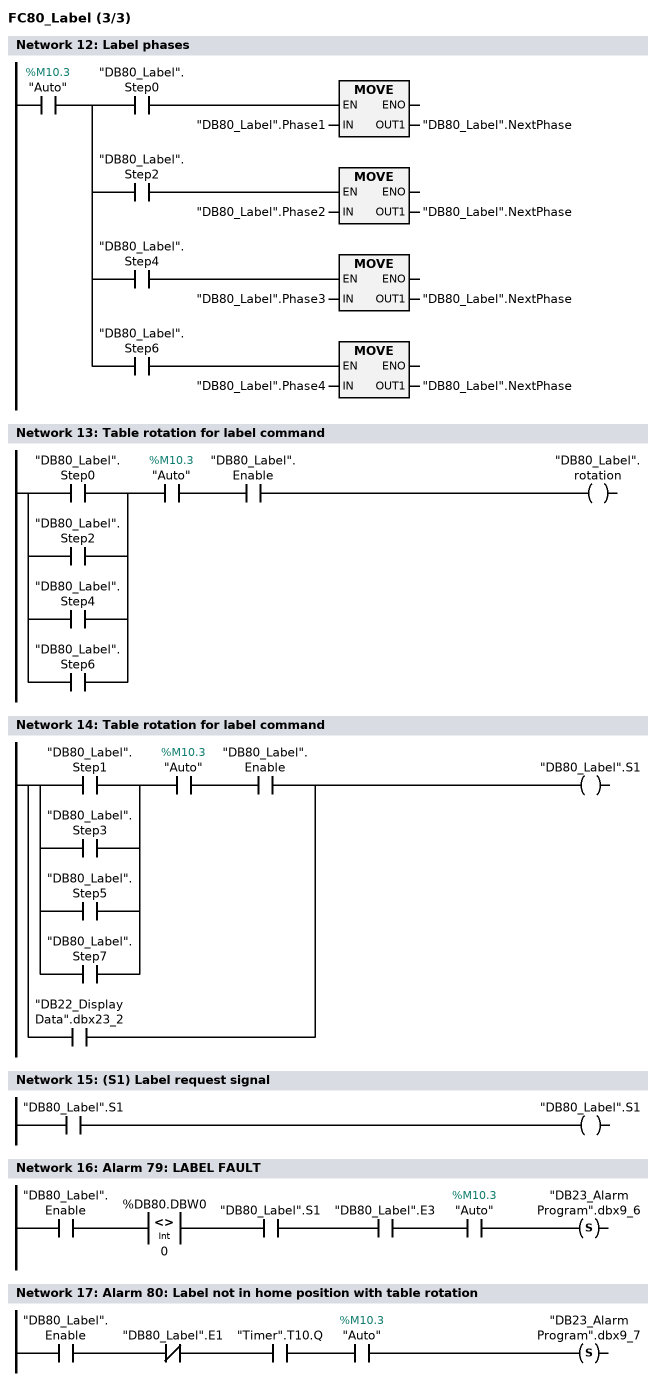
   RUNG wire#powerrail
      Contact( "Auto" )
      wire#w1
      Contact( "DB80_Label".Step0 )
      { S7_GenerateENO := "TRUE" } Move(in := "DB80_Label".Phase1, out1 => "DB80_Label".NextPhase)
   END_RUNG
   RUNG wire#w1
      Contact( "DB80_Label".Step2 )
      { S7_GenerateENO := "TRUE" } Move(in := "DB80_Label".Phase2, out1 => "DB80_Label".NextPhase)
   END_RUNG
   RUNG wire#w1
      Contact( "DB80_Label".Step4 )
      { S7_GenerateENO := "TRUE" } Move(in := "DB80_Label".Phase3, out1 => "DB80_Label".NextPhase)
   END_RUNG
   RUNG wire#w1
      Contact( "DB80_Label".Step6 )
      { S7_GenerateENO := "TRUE" } Move(in := "DB80_Label".Phase4, out1 => "DB80_Label".NextPhase)
   END_RUNG
   // the same network as SCL:
   IF "Auto" AND "DB80_Label".Step0 THEN "DB80_Label".NextPhase := "DB80_Label".Phase1; END_IF;
   IF "Auto" AND "DB80_Label".Step2 THEN "DB80_Label".NextPhase := "DB80_Label".Phase2; END_IF;
   IF "Auto" AND "DB80_Label".Step4 THEN "DB80_Label".NextPhase := "DB80_Label".Phase3; END_IF;
   IF "Auto" AND "DB80_Label".Step6 THEN "DB80_Label".NextPhase := "DB80_Label".Phase4; END_IF;
END_REGION

REGION Network 13: Table rotation for label command
   RUNG wire#powerrail
      Contact( "DB80_Label".Step0 )
      wire#w1
      Contact( "Auto" )
      Contact( "DB80_Label".Enable )
      Coil( "DB80_Label".rotation )
   END_RUNG
   RUNG wire#powerrail
      Contact( "DB80_Label".Step2 )
   END_RUNG wire#w1
   RUNG wire#powerrail
      Contact( "DB80_Label".Step4 )
   END_RUNG wire#w1
   RUNG wire#powerrail
      Contact( "DB80_Label".Step6 )
   END_RUNG wire#w1
   // the same network as SCL:
   "DB80_Label".rotation := ("DB80_Label".Step0 OR "DB80_Label".Step2 OR "DB80_Label".Step4 OR "DB80_Label".Step6) AND "Auto" AND "DB80_Label".Enable;
END_REGION

REGION Network 14: Table rotation for label command
   RUNG wire#powerrail
      Contact( "DB80_Label".Step1 )
      wire#w1
      Contact( "Auto" )
      Contact( "DB80_Label".Enable )
      wire#w2
      Coil( "DB80_Label".S1 )
   END_RUNG
   RUNG wire#powerrail
      Contact( "DB80_Label".Step3 )
   END_RUNG wire#w1
   RUNG wire#powerrail
      Contact( "DB80_Label".Step5 )
   END_RUNG wire#w1
   RUNG wire#powerrail
      Contact( "DB80_Label".Step7 )
   END_RUNG wire#w1
   RUNG wire#powerrail
      Contact( "DB22_DisplayData".dbx23_2 )
   END_RUNG wire#w2
   // the same network as SCL:
   "DB80_Label".S1 := (("DB80_Label".Step1 OR "DB80_Label".Step3 OR "DB80_Label".Step5 OR "DB80_Label".Step7) AND "Auto" AND "DB80_Label".Enable) OR "DB22_DisplayData".dbx23_2;
END_REGION

REGION Network 15: (S1) Label request signal
   RUNG wire#powerrail
      Contact( "DB80_Label".S1 )
      Coil( "DB80_Label".S1 )
   END_RUNG
   // the same network as SCL:
   "DB80_Label".S1 := "DB80_Label".S1;
END_REGION

REGION Network 16: Alarm 79: LABEL FAULT
   RUNG wire#powerrail
      Contact( "DB80_Label".Enable )
      { S7_Templates := "SrcType := Int" } NE_Contact(in1 := %DB80.DBW0, in2 := 0)
      Contact( "DB80_Label".S1 )
      Contact( "DB80_Label".E3 )
      Contact( "Auto" )
      S_Coil( "DB23_AlarmProgram".dbx9_6 )
   END_RUNG
   // the same network as SCL:
   IF "DB80_Label".Enable AND (%DB80.DBW0 <> 0) AND "DB80_Label".S1 AND "DB80_Label".E3 AND "Auto" THEN
       "DB23_AlarmProgram".dbx9_6 := TRUE;
   END_IF;
END_REGION

REGION Network 17: Alarm 80: Label not in home position with table rotation
   RUNG wire#powerrail
      Contact( "DB80_Label".Enable )
      I_Contact( "DB80_Label".E1 )
      Contact( "Timer".T10.Q )
      Contact( "Auto" )
      S_Coil( "DB23_AlarmProgram".dbx9_7 )
   END_RUNG
   // the same network as SCL:
   IF "DB80_Label".Enable AND NOT "DB80_Label".E1 AND "Timer".T10.Q AND "Auto" THEN
       "DB23_AlarmProgram".dbx9_7 := TRUE;
   END_IF;
END_REGION
END_FUNCTION

FUNCTION "FC07_FilmBroken&Test" : Void   // FC7, LAD
TITLE = Film broken or ended management
{ S7_Optimized_Access := 'FALSE' }
AUTHOR : Robopac
VERSION : 0.0
// stored: AutoNumber false, IsIECCheckEnabled false, SetENOAutomatically false, UDAEnableTagReadback false
   VAR_TEMP   // added for the SCL form of the ladder/FBD networks
      _w1 : Bool;
   END_VAR
BEGIN

REGION Network 1: Delay for test cycle
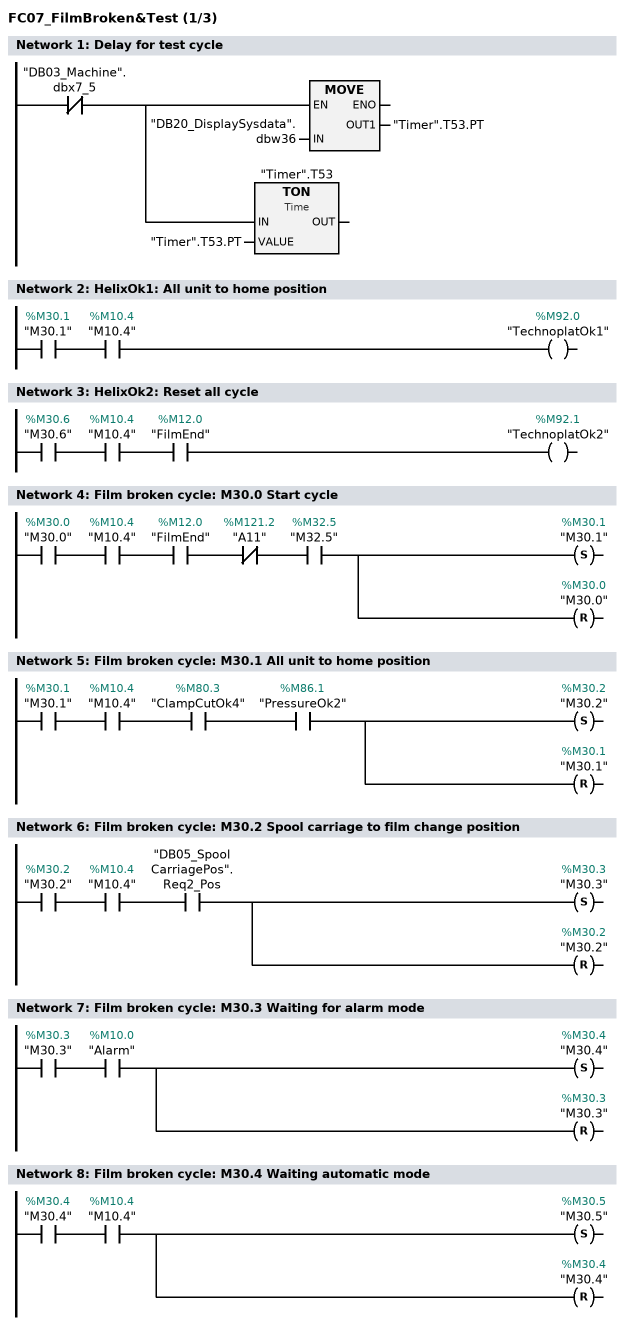
   #_w1 := NOT "DB03_Machine".dbx7_5;
   IF #_w1 THEN "Timer".T53.PT := "DB20_DisplaySysdata".dbw36; END_IF;
   "Timer".T53.TON(IN := #_w1, PT := "Timer".T53.PT);   // TON coil
END_REGION

REGION Network 2: HelixOk1: All unit to home position
   RUNG wire#powerrail
      Contact( "M30.1" )
      Contact( "M10.4" )
      Coil( "TechnoplatOk1" )
   END_RUNG
   // the same network as SCL:
   "TechnoplatOk1" := "M30.1" AND "M10.4";
END_REGION

REGION Network 3: HelixOk2: Reset all cycle
   RUNG wire#powerrail
      Contact( "M30.6" )
      Contact( "M10.4" )
      Contact( "FilmEnd" )
      Coil( "TechnoplatOk2" )
   END_RUNG
   // the same network as SCL:
   "TechnoplatOk2" := "M30.6" AND "M10.4" AND "FilmEnd";
END_REGION

REGION Network 4: Film broken cycle: M30.0 Start cycle
   RUNG wire#powerrail
      Contact( "M30.0" )
      Contact( "M10.4" )
      Contact( "FilmEnd" )
      I_Contact( "A11" )
      Contact( "M32.5" )
      wire#w1
      S_Coil( "M30.1" )
   END_RUNG
   RUNG wire#w1
      R_Coil( "M30.0" )
   END_RUNG
   // the same network as SCL:
   IF "M30.0" AND "M10.4" AND "FilmEnd" AND NOT "A11" AND "M32.5" THEN
       "M30.1" := TRUE;
       "M30.0" := FALSE;
   END_IF;
END_REGION

REGION Network 5: Film broken cycle: M30.1 All unit to home position
   RUNG wire#powerrail
      Contact( "M30.1" )
      Contact( "M10.4" )
      Contact( "ClampCutOk4" )
      Contact( "PressureOk2" )
      wire#w1
      S_Coil( "M30.2" )
   END_RUNG
   RUNG wire#w1
      R_Coil( "M30.1" )
   END_RUNG
   // the same network as SCL:
   IF "M30.1" AND "M10.4" AND "ClampCutOk4" AND "PressureOk2" THEN
       "M30.2" := TRUE;
       "M30.1" := FALSE;
   END_IF;
END_REGION

REGION Network 6: Film broken cycle: M30.2 Spool carriage to film change position
   RUNG wire#powerrail
      Contact( "M30.2" )
      Contact( "M10.4" )
      Contact( "DB05_SpoolCarriagePos".Req2_Pos )
      wire#w1
      S_Coil( "M30.3" )
   END_RUNG
   RUNG wire#w1
      R_Coil( "M30.2" )
   END_RUNG
   // the same network as SCL:
   IF "M30.2" AND "M10.4" AND "DB05_SpoolCarriagePos".Req2_Pos THEN
       "M30.3" := TRUE;
       "M30.2" := FALSE;
   END_IF;
END_REGION

REGION Network 7: Film broken cycle: M30.3 Waiting for alarm mode
   RUNG wire#powerrail
      Contact( "M30.3" )
      Contact( "Alarm" )
      wire#w1
      S_Coil( "M30.4" )
   END_RUNG
   RUNG wire#w1
      R_Coil( "M30.3" )
   END_RUNG
   // the same network as SCL:
   IF "M30.3" AND "Alarm" THEN
       "M30.4" := TRUE;
       "M30.3" := FALSE;
   END_IF;
END_REGION

REGION Network 8: Film broken cycle: M30.4 Waiting automatic mode
   RUNG wire#powerrail
      Contact( "M30.4" )
      Contact( "M10.4" )
      wire#w1
      S_Coil( "M30.5" )
   END_RUNG
   RUNG wire#w1
      R_Coil( "M30.4" )
   END_RUNG
   // the same network as SCL:
   IF "M30.4" AND "M10.4" THEN
       "M30.5" := TRUE;
       "M30.4" := FALSE;
   END_IF;
END_REGION

REGION Network 9: Film broken cycle: M30.5 Spool carriage downward
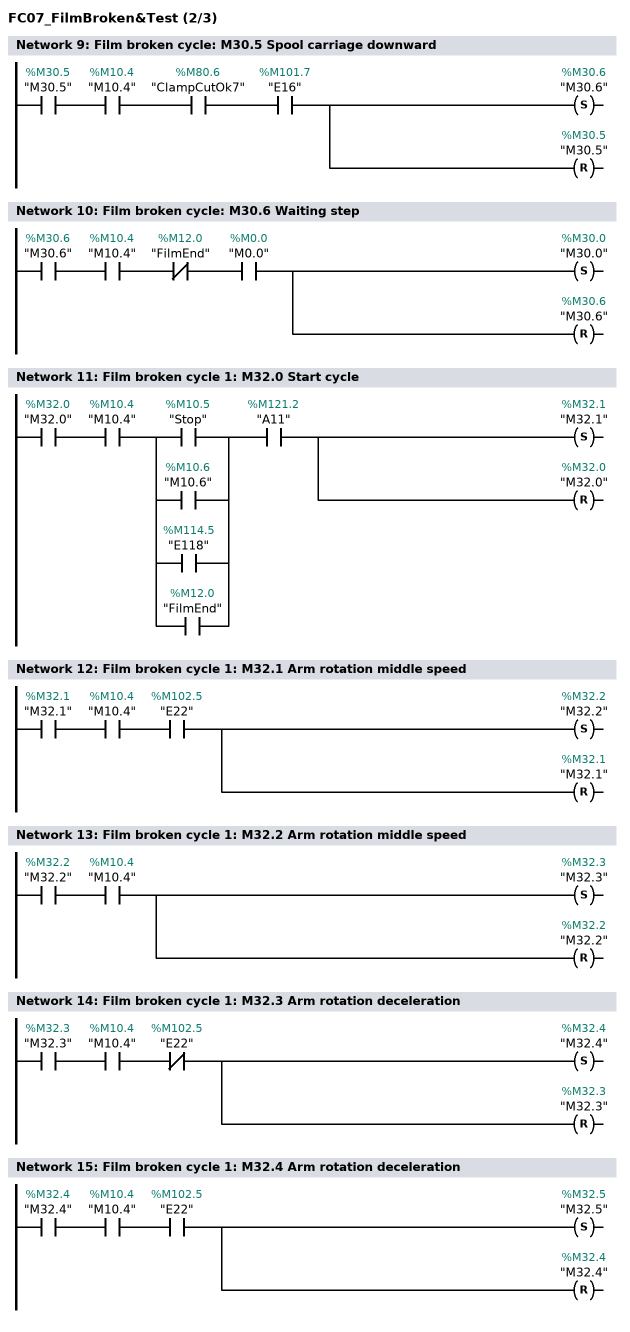
   RUNG wire#powerrail
      Contact( "M30.5" )
      Contact( "M10.4" )
      Contact( "ClampCutOk7" )
      Contact( "E16" )
      wire#w1
      S_Coil( "M30.6" )
   END_RUNG
   RUNG wire#w1
      R_Coil( "M30.5" )
   END_RUNG
   // the same network as SCL:
   IF "M30.5" AND "M10.4" AND "ClampCutOk7" AND "E16" THEN
       "M30.6" := TRUE;
       "M30.5" := FALSE;
   END_IF;
END_REGION

REGION Network 10: Film broken cycle: M30.6 Waiting step
   RUNG wire#powerrail
      Contact( "M30.6" )
      Contact( "M10.4" )
      I_Contact( "FilmEnd" )
      Contact( "M0.0" )
      wire#w1
      S_Coil( "M30.0" )
   END_RUNG
   RUNG wire#w1
      R_Coil( "M30.6" )
   END_RUNG
   // the same network as SCL:
   IF "M30.6" AND "M10.4" AND NOT "FilmEnd" AND "M0.0" THEN
       "M30.0" := TRUE;
       "M30.6" := FALSE;
   END_IF;
END_REGION

REGION Network 11: Film broken cycle 1: M32.0 Start cycle
   RUNG wire#powerrail
      Contact( "M32.0" )
      Contact( "M10.4" )
      wire#w1
      Contact( "Stop" )
      wire#w2
      Contact( "A11" )
      wire#w3
      S_Coil( "M32.1" )
   END_RUNG
   RUNG wire#w1
      Contact( "M10.6" )
   END_RUNG wire#w2
   RUNG wire#w1
      Contact( "E118" )
   END_RUNG wire#w2
   RUNG wire#w1
      Contact( "FilmEnd" )
   END_RUNG wire#w2
   RUNG wire#w3
      R_Coil( "M32.0" )
   END_RUNG
   // the same network as SCL:
   IF "M32.0" AND "M10.4" AND ("Stop" OR "M10.6" OR "E118" OR "FilmEnd") AND "A11" THEN
       "M32.1" := TRUE;
       "M32.0" := FALSE;
   END_IF;
END_REGION

REGION Network 12: Film broken cycle 1: M32.1 Arm rotation middle speed
   RUNG wire#powerrail
      Contact( "M32.1" )
      Contact( "M10.4" )
      Contact( "E22" )
      wire#w1
      S_Coil( "M32.2" )
   END_RUNG
   RUNG wire#w1
      R_Coil( "M32.1" )
   END_RUNG
   // the same network as SCL:
   IF "M32.1" AND "M10.4" AND "E22" THEN
       "M32.2" := TRUE;
       "M32.1" := FALSE;
   END_IF;
END_REGION

REGION Network 13: Film broken cycle 1: M32.2 Arm rotation middle speed
   RUNG wire#powerrail
      Contact( "M32.2" )
      Contact( "M10.4" )
      wire#w1
      S_Coil( "M32.3" )
   END_RUNG
   RUNG wire#w1
      R_Coil( "M32.2" )
   END_RUNG
   // the same network as SCL:
   IF "M32.2" AND "M10.4" THEN
       "M32.3" := TRUE;
       "M32.2" := FALSE;
   END_IF;
END_REGION

REGION Network 14: Film broken cycle 1: M32.3 Arm rotation deceleration
   RUNG wire#powerrail
      Contact( "M32.3" )
      Contact( "M10.4" )
      I_Contact( "E22" )
      wire#w1
      S_Coil( "M32.4" )
   END_RUNG
   RUNG wire#w1
      R_Coil( "M32.3" )
   END_RUNG
   // the same network as SCL:
   IF "M32.3" AND "M10.4" AND NOT "E22" THEN
       "M32.4" := TRUE;
       "M32.3" := FALSE;
   END_IF;
END_REGION

REGION Network 15: Film broken cycle 1: M32.4 Arm rotation deceleration
   RUNG wire#powerrail
      Contact( "M32.4" )
      Contact( "M10.4" )
      Contact( "E22" )
      wire#w1
      S_Coil( "M32.5" )
   END_RUNG
   RUNG wire#w1
      R_Coil( "M32.4" )
   END_RUNG
   // the same network as SCL:
   IF "M32.4" AND "M10.4" AND "E22" THEN
       "M32.5" := TRUE;
       "M32.4" := FALSE;
   END_IF;
END_REGION

REGION Network 16: Film broken cycle 1: M32.5 Waiting step
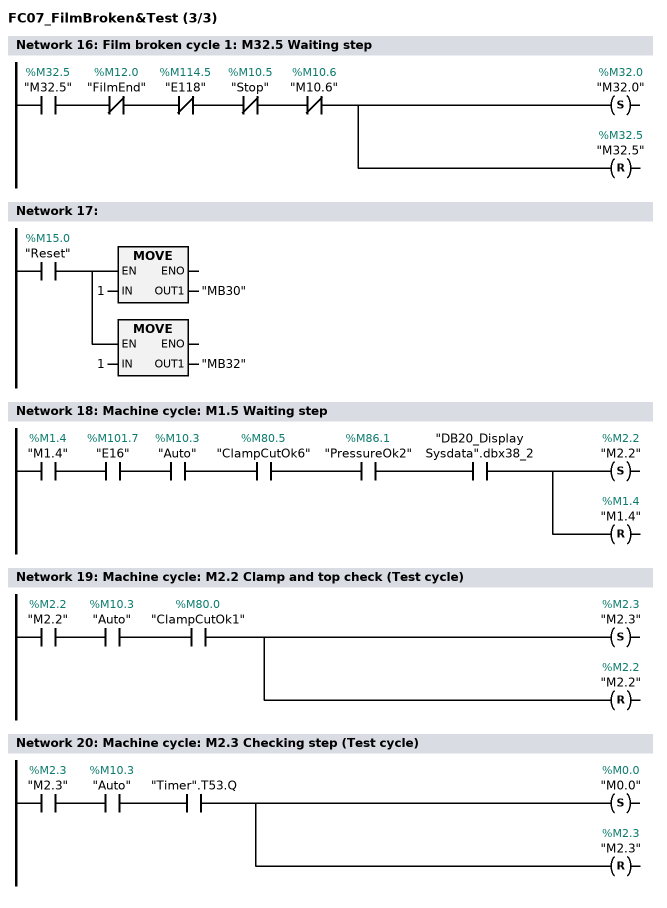
   RUNG wire#powerrail
      Contact( "M32.5" )
      I_Contact( "FilmEnd" )
      I_Contact( "E118" )
      I_Contact( "Stop" )
      I_Contact( "M10.6" )
      wire#w1
      S_Coil( "M32.0" )
   END_RUNG
   RUNG wire#w1
      R_Coil( "M32.5" )
   END_RUNG
   // the same network as SCL:
   IF "M32.5" AND NOT "FilmEnd" AND NOT "E118" AND NOT "Stop" AND NOT "M10.6" THEN
       "M32.0" := TRUE;
       "M32.5" := FALSE;
   END_IF;
END_REGION

REGION Network 17
   RUNG wire#powerrail
      Contact( "Reset" )
      wire#w1
      { S7_GenerateENO := "TRUE" } Move(in := 1, out1 => "MB30")
   END_RUNG
   RUNG wire#w1
      { S7_GenerateENO := "TRUE" } Move(in := 1, out1 => "MB32")
   END_RUNG
   // the same network as SCL:
   IF "Reset" THEN
       "MB30" := 1;
       "MB32" := 1;
   END_IF;
END_REGION

REGION Network 18: Machine cycle: M1.5 Waiting step
   RUNG wire#powerrail
      Contact( "M1.4" )
      Contact( "E16" )
      Contact( "Auto" )
      Contact( "ClampCutOk6" )
      Contact( "PressureOk2" )
      Contact( "DB20_DisplaySysdata".dbx38_2 )
      wire#w1
      S_Coil( "M2.2" )
   END_RUNG
   RUNG wire#w1
      R_Coil( "M1.4" )
   END_RUNG
   // the same network as SCL:
   IF "M1.4" AND "E16" AND "Auto" AND "ClampCutOk6" AND "PressureOk2" AND "DB20_DisplaySysdata".dbx38_2 THEN
       "M2.2" := TRUE;
       "M1.4" := FALSE;
   END_IF;
END_REGION

REGION Network 19: Machine cycle: M2.2 Clamp and top check (Test cycle)
   RUNG wire#powerrail
      Contact( "M2.2" )
      Contact( "Auto" )
      Contact( "ClampCutOk1" )
      wire#w1
      S_Coil( "M2.3" )
   END_RUNG
   RUNG wire#w1
      R_Coil( "M2.2" )
   END_RUNG
   // the same network as SCL:
   IF "M2.2" AND "Auto" AND "ClampCutOk1" THEN
       "M2.3" := TRUE;
       "M2.2" := FALSE;
   END_IF;
END_REGION

REGION Network 20: Machine cycle: M2.3 Checking step (Test cycle)
   RUNG wire#powerrail
      Contact( "M2.3" )
      Contact( "Auto" )
      Contact( "Timer".T53.Q )
      wire#w1
      S_Coil( "M0.0" )
   END_RUNG
   RUNG wire#w1
      R_Coil( "M2.3" )
   END_RUNG
   // the same network as SCL:
   IF "M2.3" AND "Auto" AND "Timer".T53.Q THEN
       "M0.0" := TRUE;
       "M2.3" := FALSE;
   END_IF;
END_REGION
END_FUNCTION

FUNCTION "FC45_PrestretchPGSM_PGSA" : Void   // FC45, LAD
TITLE = Prestretch PGSM and PGSA management (HS30, Helix One)
{ S7_Optimized_Access := 'FALSE' }
AUTHOR : Robopac
VERSION : 0.0
// stored: AutoNumber false, IsIECCheckEnabled false, SetENOAutomatically false, UDAEnableTagReadback false
   VAR_TEMP
      TempInt : Int;
      TempDint : DInt;
      TempDint_2 : DInt;
      TiroStepTemp : Int;
      TiroFineTemp : Int;
   END_VAR
   VAR_TEMP   // added for the SCL form of the ladder/FBD networks
      _w1 : Bool;
      _w2 : Bool;
      _w3 : Bool;
      _w4 : Bool;
      _w5 : Bool;
      _w6 : Bool;
      _w7 : Bool;
   END_VAR
BEGIN

REGION Network 1: Film broken delay for spool carriage
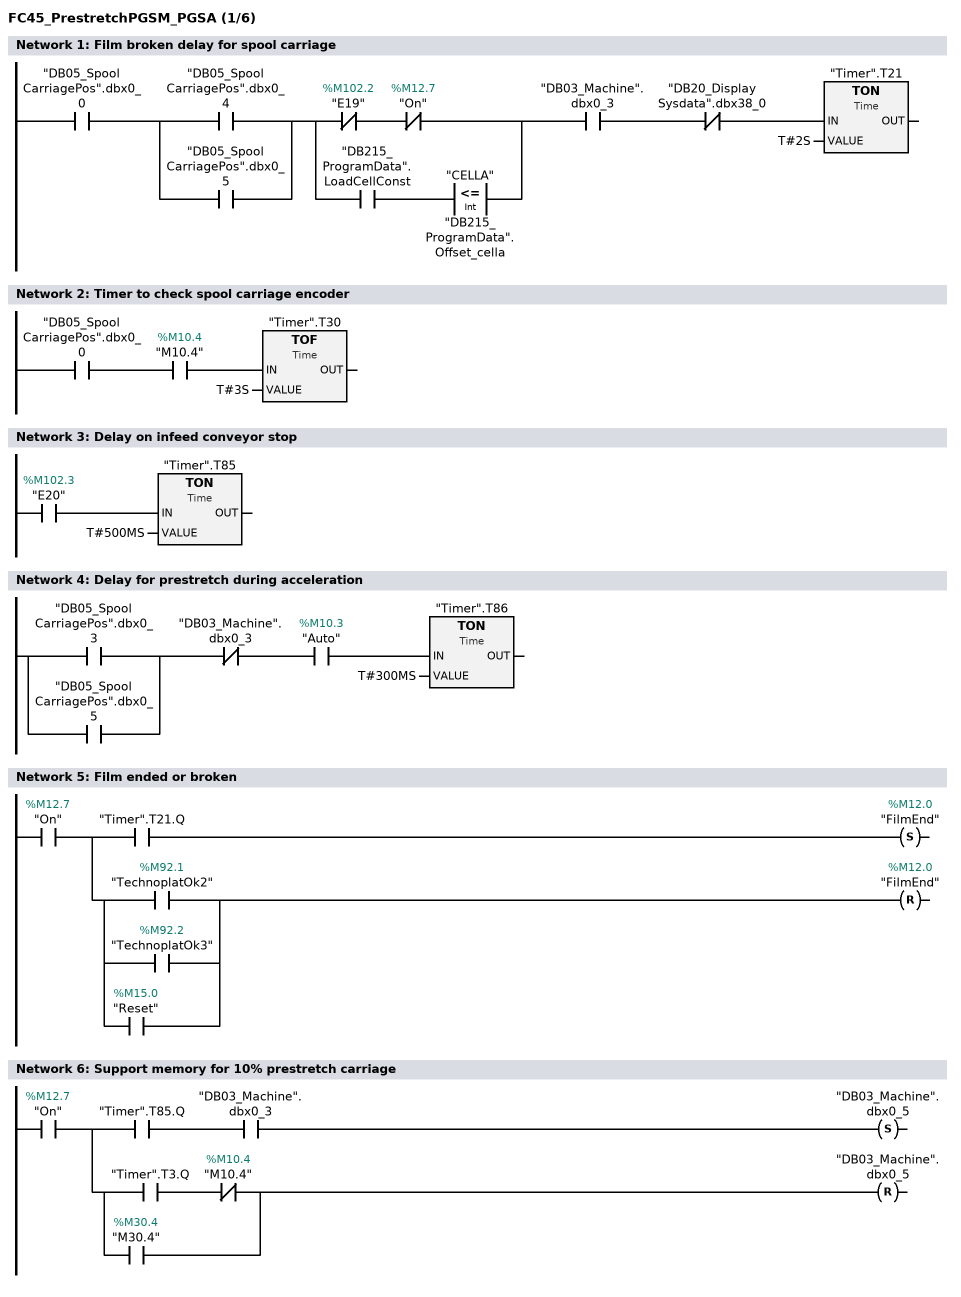
   "Timer".T21.TON(IN := "DB05_SpoolCarriagePos".dbx0_0 AND ("DB05_SpoolCarriagePos".dbx0_4 OR "DB05_SpoolCarriagePos".dbx0_5) AND ((NOT "E19" AND NOT "On") OR ("DB215_ProgramData".LoadCellConst AND ("CELLA" <= "DB215_ProgramData".Offset_cella))) AND "DB03_Machine".dbx0_3 AND NOT "DB20_DisplaySysdata".dbx38_0, PT := T#2S);   // TON coil
END_REGION

REGION Network 2: Timer to check spool carriage encoder
   "Timer".T30.TOF(IN := "DB05_SpoolCarriagePos".dbx0_0 AND "M10.4", PT := T#3S);   // TOF coil
END_REGION

REGION Network 3: Delay on infeed conveyor stop
   "Timer".T85.TON(IN := "E20", PT := T#500MS);   // TON coil
END_REGION

REGION Network 4: Delay for prestretch during acceleration
   "Timer".T86.TON(IN := ("DB05_SpoolCarriagePos".dbx0_3 OR "DB05_SpoolCarriagePos".dbx0_5) AND NOT "DB03_Machine".dbx0_3 AND "Auto", PT := T#300MS);   // TON coil
END_REGION

REGION Network 5: Film ended or broken
   RUNG wire#powerrail
      Contact( "On" )
      wire#w1
      Contact( "Timer".T21.Q )
      S_Coil( "FilmEnd" )
   END_RUNG
   RUNG wire#w1
      Contact( "TechnoplatOk2" )
      wire#w2
      R_Coil( "FilmEnd" )
   END_RUNG
   RUNG wire#w1
      Contact( "TechnoplatOk3" )
   END_RUNG wire#w2
   RUNG wire#w1
      Contact( "Reset" )
   END_RUNG wire#w2
   // the same network as SCL:
   IF "On" AND "Timer".T21.Q THEN "FilmEnd" := TRUE; END_IF;
   IF "On" AND ("TechnoplatOk2" OR "TechnoplatOk3" OR "Reset") THEN "FilmEnd" := FALSE; END_IF;
END_REGION

REGION Network 6: Support memory for 10% prestretch carriage
   RUNG wire#powerrail
      Contact( "On" )
      wire#w1
      Contact( "Timer".T85.Q )
      Contact( "DB03_Machine".dbx0_3 )
      S_Coil( "DB03_Machine".dbx0_5 )
   END_RUNG
   RUNG wire#w1
      Contact( "Timer".T3.Q )
      I_Contact( "M10.4" )
      wire#w2
      R_Coil( "DB03_Machine".dbx0_5 )
   END_RUNG
   RUNG wire#w1
      Contact( "M30.4" )
   END_RUNG wire#w2
   // the same network as SCL:
   IF "On" AND "Timer".T85.Q AND "DB03_Machine".dbx0_3 THEN "DB03_Machine".dbx0_5 := TRUE; END_IF;
   IF "On" AND (("Timer".T3.Q AND NOT "M10.4") OR "M30.4") THEN "DB03_Machine".dbx0_5 := FALSE; END_IF;
END_REGION

REGION Network 7: Support memory for prestretch PGSM or PGSA
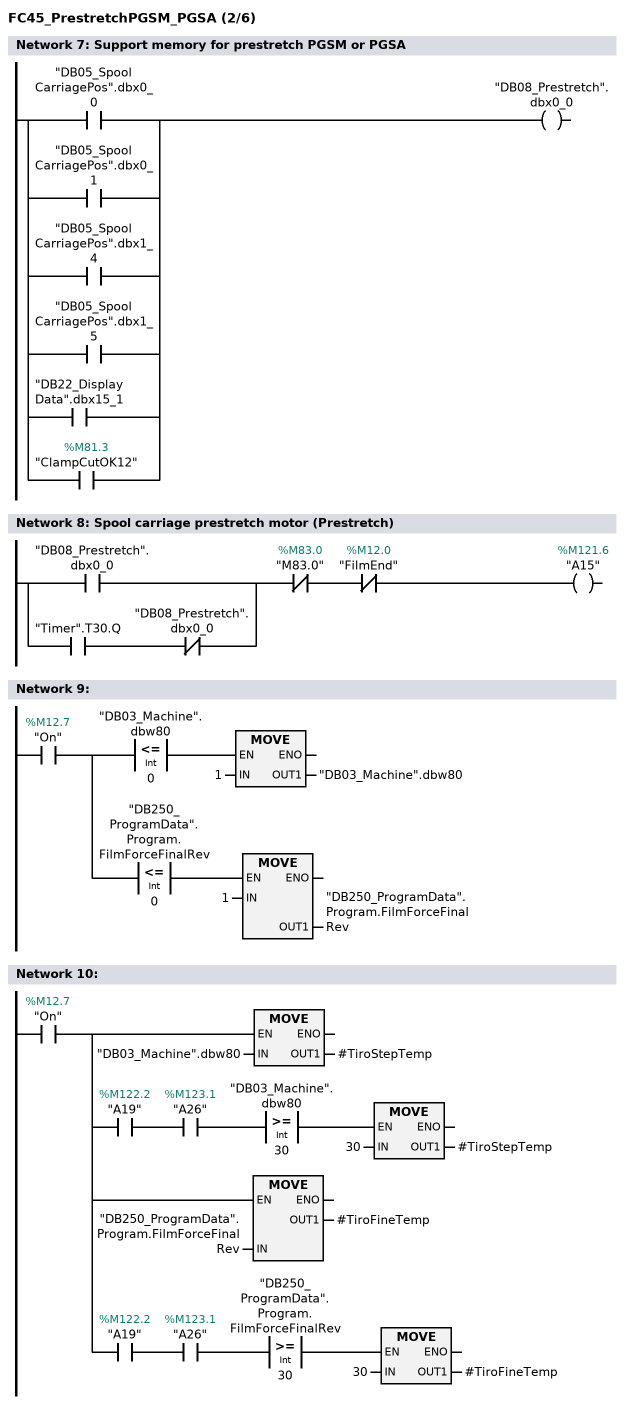
   RUNG wire#powerrail
      Contact( "DB05_SpoolCarriagePos".dbx0_0 )
      wire#w1
      Coil( "DB08_Prestretch".dbx0_0 )
   END_RUNG
   RUNG wire#powerrail
      Contact( "DB05_SpoolCarriagePos".dbx0_1 )
   END_RUNG wire#w1
   RUNG wire#powerrail
      Contact( "DB05_SpoolCarriagePos".dbx1_4 )
   END_RUNG wire#w1
   RUNG wire#powerrail
      Contact( "DB05_SpoolCarriagePos".dbx1_5 )
   END_RUNG wire#w1
   RUNG wire#powerrail
      Contact( "DB22_DisplayData".dbx15_1 )
   END_RUNG wire#w1
   RUNG wire#powerrail
      Contact( "ClampCutOK12" )
   END_RUNG wire#w1
   // the same network as SCL:
   "DB08_Prestretch".dbx0_0 := "DB05_SpoolCarriagePos".dbx0_0 OR "DB05_SpoolCarriagePos".dbx0_1 OR "DB05_SpoolCarriagePos".dbx1_4 OR "DB05_SpoolCarriagePos".dbx1_5 OR "DB22_DisplayData".dbx15_1 OR "ClampCutOK12";
END_REGION

REGION Network 8: Spool carriage prestretch motor (Prestretch)
   RUNG wire#powerrail
      Contact( "DB08_Prestretch".dbx0_0 )
      wire#w1
      I_Contact( "M83.0" )
      I_Contact( "FilmEnd" )
      Coil( "A15" )
   END_RUNG
   RUNG wire#powerrail
      Contact( "Timer".T30.Q )
      I_Contact( "DB08_Prestretch".dbx0_0 )
   END_RUNG wire#w1
   // the same network as SCL:
   "A15" := ("DB08_Prestretch".dbx0_0 OR ("Timer".T30.Q AND NOT "DB08_Prestretch".dbx0_0)) AND NOT "M83.0" AND NOT "FilmEnd";
END_REGION

REGION Network 9
   RUNG wire#powerrail
      Contact( "On" )
      wire#w1
      { S7_Templates := "SrcType := Int" } LE_Contact(in1 := "DB03_Machine".dbw80, in2 := 0)
      { S7_GenerateENO := "TRUE" } Move(in := 1, out1 => "DB03_Machine".dbw80)
   END_RUNG
   RUNG wire#w1
      { S7_Templates := "SrcType := Int" } LE_Contact(in1 := "DB250_ProgramData".Program.FilmForceFinalRev, in2 := 0)
      { S7_GenerateENO := "TRUE" } Move(in := 1, out1 => "DB250_ProgramData".Program.FilmForceFinalRev)
   END_RUNG
   // the same network as SCL:
   IF "On" AND ("DB03_Machine".dbw80 <= 0) THEN "DB03_Machine".dbw80 := 1; END_IF;
   IF "On" AND ("DB250_ProgramData".Program.FilmForceFinalRev <= 0) THEN
       "DB250_ProgramData".Program.FilmForceFinalRev := 1;
   END_IF;
END_REGION

REGION Network 10
   RUNG wire#powerrail
      Contact( "On" )
      wire#w1
      { S7_GenerateENO := "TRUE" } Move(in := "DB03_Machine".dbw80, out1 => #TiroStepTemp)
   END_RUNG
   RUNG wire#w1
      Contact( "A19" )
      Contact( "A26" )
      { S7_Templates := "SrcType := Int" } GE_Contact(in1 := "DB03_Machine".dbw80, in2 := 30)
      { S7_GenerateENO := "TRUE" } Move(in := 30, out1 => #TiroStepTemp)
   END_RUNG
   RUNG wire#w1
      { S7_GenerateENO := "TRUE" } Move(in := "DB250_ProgramData".Program.FilmForceFinalRev, out1 => #TiroFineTemp)
   END_RUNG
   RUNG wire#w1
      Contact( "A19" )
      Contact( "A26" )
      { S7_Templates := "SrcType := Int" } GE_Contact(in1 := "DB250_ProgramData".Program.FilmForceFinalRev, in2 := 30)
      { S7_GenerateENO := "TRUE" } Move(in := 30, out1 => #TiroFineTemp)
   END_RUNG
   // the same network as SCL:
   IF "On" THEN #TiroStepTemp := "DB03_Machine".dbw80; END_IF;
   IF "On" AND "A19" AND "A26" AND ("DB03_Machine".dbw80 >= 30) THEN #TiroStepTemp := 30; END_IF;
   IF "On" THEN #TiroFineTemp := "DB250_ProgramData".Program.FilmForceFinalRev; END_IF;
   IF "On" AND "A19" AND "A26" AND ("DB250_ProgramData".Program.FilmForceFinalRev >= 30) THEN
       #TiroFineTemp := 30;
   END_IF;
END_REGION

REGION Network 11
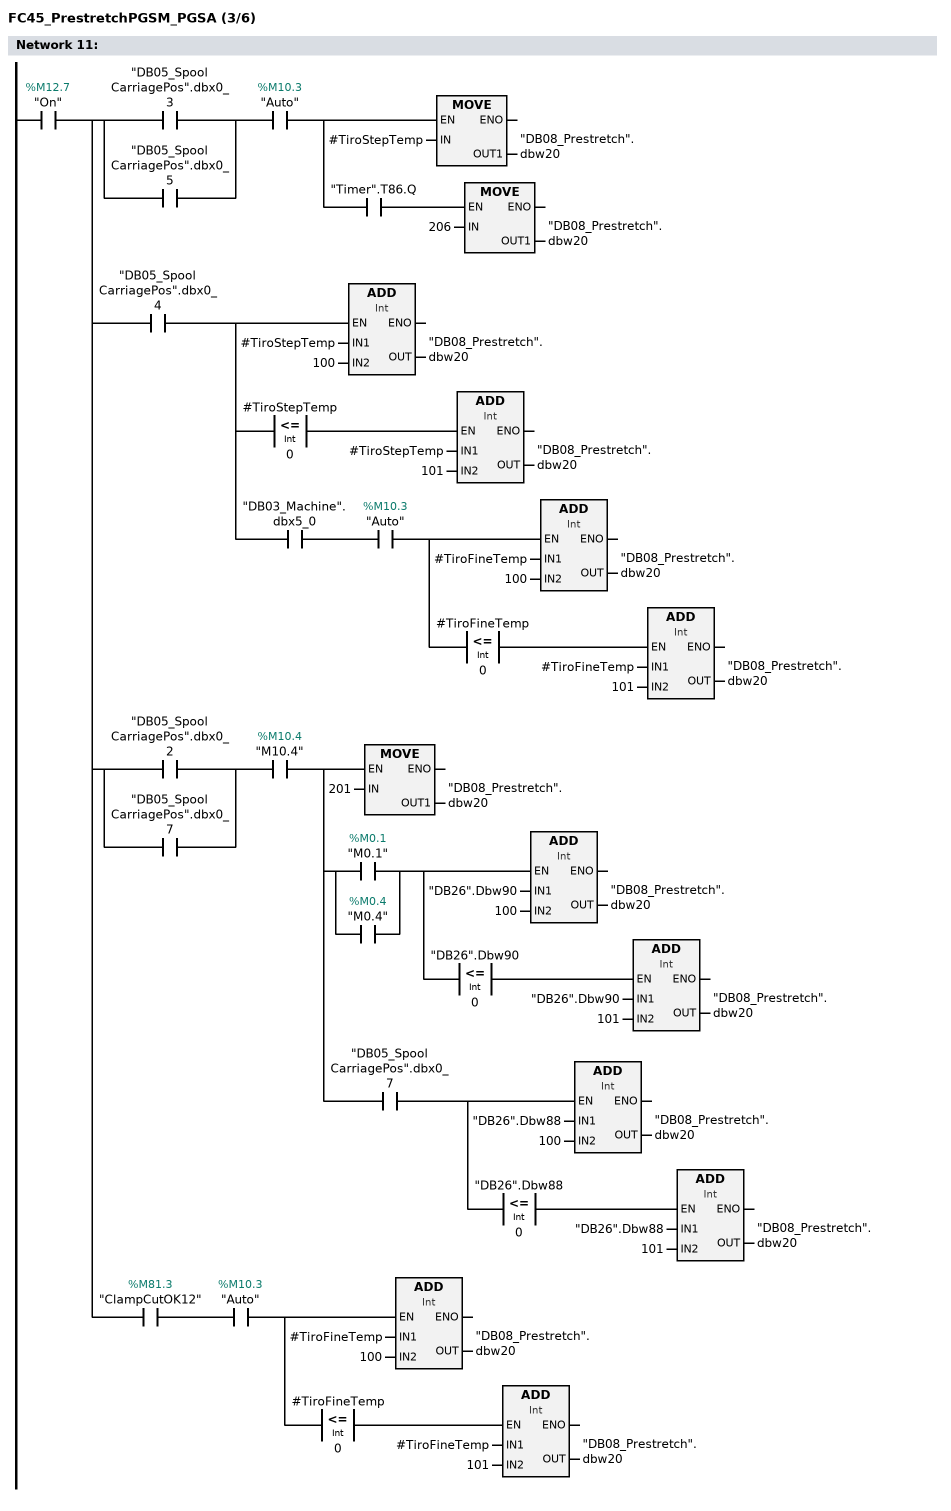
   RUNG wire#powerrail
      Contact( "On" )
      wire#w1
      Contact( "DB05_SpoolCarriagePos".dbx0_3 )
      wire#w2
      Contact( "Auto" )
      wire#w3
      { S7_GenerateENO := "TRUE" } Move(in := #TiroStepTemp, out1 => "DB08_Prestretch".dbw20)
   END_RUNG
   RUNG wire#w1
      Contact( "DB05_SpoolCarriagePos".dbx0_5 )
   END_RUNG wire#w2
   RUNG wire#w3
      Contact( "Timer".T86.Q )
      { S7_GenerateENO := "TRUE" } Move(in := 206, out1 => "DB08_Prestretch".dbw20)
   END_RUNG
   RUNG wire#w1
      Contact( "DB05_SpoolCarriagePos".dbx0_4 )
      wire#w4
      { S7_Templates := "SrcType := Int"; S7_GenerateENO := "TRUE" } Add(in1 := #TiroStepTemp, in2 := 100, out => "DB08_Prestretch".dbw20)
   END_RUNG
   RUNG wire#w4
      { S7_Templates := "SrcType := Int" } LE_Contact(in1 := #TiroStepTemp, in2 := 0)
      { S7_Templates := "SrcType := Int"; S7_GenerateENO := "TRUE" } Add(in1 := #TiroStepTemp, in2 := 101, out => "DB08_Prestretch".dbw20)
   END_RUNG
   RUNG wire#w4
      Contact( "DB03_Machine".dbx5_0 )
      Contact( "Auto" )
      wire#w5
      { S7_Templates := "SrcType := Int"; S7_GenerateENO := "TRUE" } Add(in1 := #TiroFineTemp, in2 := 100, out => "DB08_Prestretch".dbw20)
   END_RUNG
   RUNG wire#w5
      { S7_Templates := "SrcType := Int" } LE_Contact(in1 := #TiroFineTemp, in2 := 0)
      { S7_Templates := "SrcType := Int"; S7_GenerateENO := "TRUE" } Add(in1 := #TiroFineTemp, in2 := 101, out => "DB08_Prestretch".dbw20)
   END_RUNG
   RUNG wire#w1
      Contact( "DB05_SpoolCarriagePos".dbx0_2 )
      wire#w6
      Contact( "M10.4" )
      wire#w7
      { S7_GenerateENO := "TRUE" } Move(in := 201, out1 => "DB08_Prestretch".dbw20)
   END_RUNG
   RUNG wire#w1
      Contact( "DB05_SpoolCarriagePos".dbx0_7 )
   END_RUNG wire#w6
   RUNG wire#w7
      Contact( "M0.1" )
      wire#w8
      { S7_Templates := "SrcType := Int"; S7_GenerateENO := "TRUE" } Add(in1 := "DB26".Dbw90, in2 := 100, out => "DB08_Prestretch".dbw20)
   END_RUNG
   RUNG wire#w7
      Contact( "M0.4" )
   END_RUNG wire#w8
   RUNG wire#w8
      { S7_Templates := "SrcType := Int" } LE_Contact(in1 := "DB26".Dbw90, in2 := 0)
      { S7_Templates := "SrcType := Int"; S7_GenerateENO := "TRUE" } Add(in1 := "DB26".Dbw90, in2 := 101, out => "DB08_Prestretch".dbw20)
   END_RUNG
   RUNG wire#w7
      Contact( "DB05_SpoolCarriagePos".dbx0_7 )
      wire#w9
      { S7_Templates := "SrcType := Int"; S7_GenerateENO := "TRUE" } Add(in1 := "DB26".Dbw88, in2 := 100, out => "DB08_Prestretch".dbw20)
   END_RUNG
   RUNG wire#w9
      { S7_Templates := "SrcType := Int" } LE_Contact(in1 := "DB26".Dbw88, in2 := 0)
      { S7_Templates := "SrcType := Int"; S7_GenerateENO := "TRUE" } Add(in1 := "DB26".Dbw88, in2 := 101, out => "DB08_Prestretch".dbw20)
   END_RUNG
   RUNG wire#w1
      Contact( "ClampCutOK12" )
      Contact( "Auto" )
      wire#w10
      { S7_Templates := "SrcType := Int"; S7_GenerateENO := "TRUE" } Add(in1 := #TiroFineTemp, in2 := 100, out => "DB08_Prestretch".dbw20)
   END_RUNG
   RUNG wire#w10
      { S7_Templates := "SrcType := Int" } LE_Contact(in1 := #TiroFineTemp, in2 := 0)
      { S7_Templates := "SrcType := Int"; S7_GenerateENO := "TRUE" } Add(in1 := #TiroFineTemp, in2 := 101, out => "DB08_Prestretch".dbw20)
   END_RUNG
   // the same network as SCL:
   #_w1 := "On" AND ("DB05_SpoolCarriagePos".dbx0_3 OR "DB05_SpoolCarriagePos".dbx0_5) AND "Auto";
   IF #_w1 THEN "DB08_Prestretch".dbw20 := #TiroStepTemp; END_IF;
   IF #_w1 AND "Timer".T86.Q THEN "DB08_Prestretch".dbw20 := 206; END_IF;
   #_w2 := "On" AND "DB05_SpoolCarriagePos".dbx0_4;
   IF #_w2 THEN "DB08_Prestretch".dbw20 := #TiroStepTemp + 100; END_IF;
   IF #_w2 AND (#TiroStepTemp <= 0) THEN "DB08_Prestretch".dbw20 := #TiroStepTemp + 101; END_IF;
   #_w3 := #_w2 AND "DB03_Machine".dbx5_0 AND "Auto";
   IF #_w3 THEN "DB08_Prestretch".dbw20 := #TiroFineTemp + 100; END_IF;
   IF #_w3 AND (#TiroFineTemp <= 0) THEN "DB08_Prestretch".dbw20 := #TiroFineTemp + 101; END_IF;
   #_w4 := "On" AND ("DB05_SpoolCarriagePos".dbx0_2 OR "DB05_SpoolCarriagePos".dbx0_7) AND "M10.4";
   IF #_w4 THEN "DB08_Prestretch".dbw20 := 201; END_IF;
   #_w5 := #_w4 AND ("M0.1" OR "M0.4");
   IF #_w5 THEN "DB08_Prestretch".dbw20 := "DB26".Dbw90 + 100; END_IF;
   IF #_w5 AND ("DB26".Dbw90 <= 0) THEN "DB08_Prestretch".dbw20 := "DB26".Dbw90 + 101; END_IF;
   #_w6 := #_w4 AND "DB05_SpoolCarriagePos".dbx0_7;
   IF #_w6 THEN "DB08_Prestretch".dbw20 := "DB26".Dbw88 + 100; END_IF;
   IF #_w6 AND ("DB26".Dbw88 <= 0) THEN "DB08_Prestretch".dbw20 := "DB26".Dbw88 + 101; END_IF;
   #_w7 := "On" AND "ClampCutOK12" AND "Auto";
   IF #_w7 THEN "DB08_Prestretch".dbw20 := #TiroFineTemp + 100; END_IF;
   IF #_w7 AND (#TiroFineTemp <= 0) THEN "DB08_Prestretch".dbw20 := #TiroFineTemp + 101; END_IF;
END_REGION

REGION Network 12
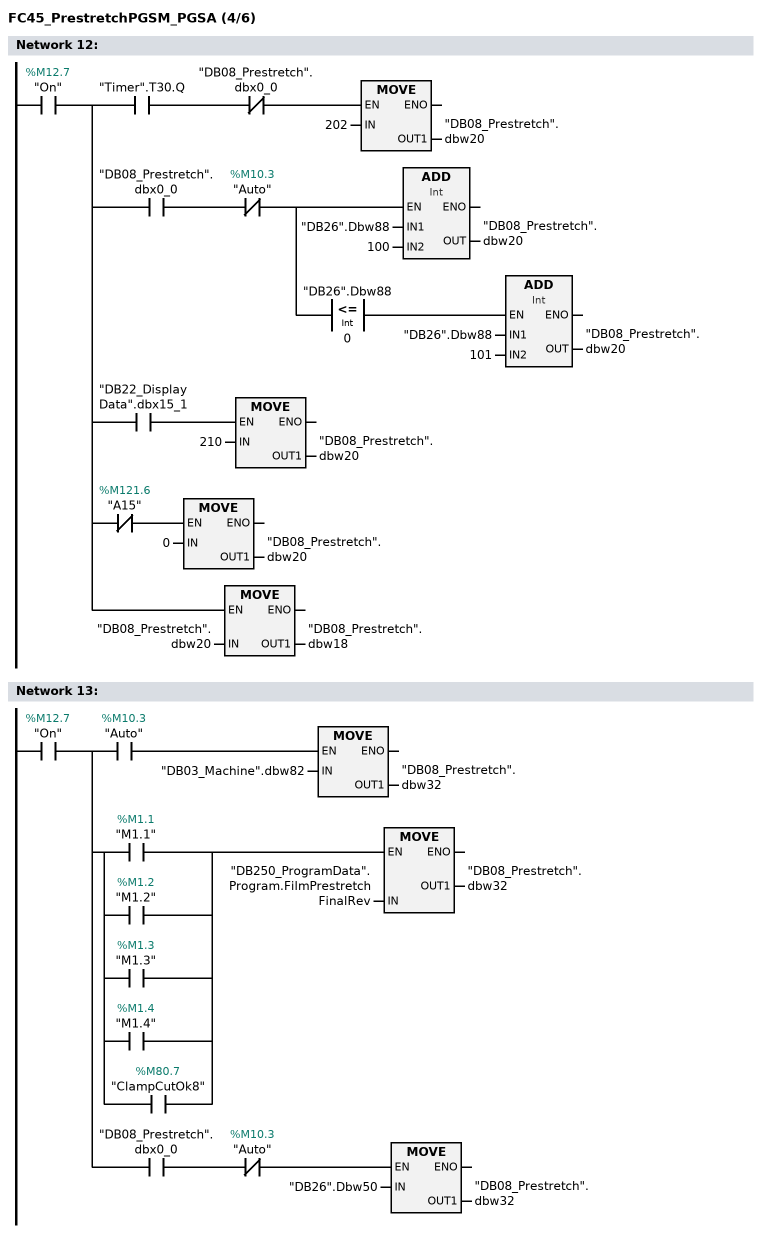
   RUNG wire#powerrail
      Contact( "On" )
      wire#w1
      Contact( "Timer".T30.Q )
      I_Contact( "DB08_Prestretch".dbx0_0 )
      { S7_GenerateENO := "TRUE" } Move(in := 202, out1 => "DB08_Prestretch".dbw20)
   END_RUNG
   RUNG wire#w1
      Contact( "DB08_Prestretch".dbx0_0 )
      I_Contact( "Auto" )
      wire#w2
      { S7_Templates := "SrcType := Int"; S7_GenerateENO := "TRUE" } Add(in1 := "DB26".Dbw88, in2 := 100, out => "DB08_Prestretch".dbw20)
   END_RUNG
   RUNG wire#w2
      { S7_Templates := "SrcType := Int" } LE_Contact(in1 := "DB26".Dbw88, in2 := 0)
      { S7_Templates := "SrcType := Int"; S7_GenerateENO := "TRUE" } Add(in1 := "DB26".Dbw88, in2 := 101, out => "DB08_Prestretch".dbw20)
   END_RUNG
   RUNG wire#w1
      Contact( "DB22_DisplayData".dbx15_1 )
      { S7_GenerateENO := "TRUE" } Move(in := 210, out1 => "DB08_Prestretch".dbw20)
   END_RUNG
   RUNG wire#w1
      I_Contact( "A15" )
      { S7_GenerateENO := "TRUE" } Move(in := 0, out1 => "DB08_Prestretch".dbw20)
   END_RUNG
   RUNG wire#w1
      { S7_GenerateENO := "TRUE" } Move(in := "DB08_Prestretch".dbw20, out1 => "DB08_Prestretch".dbw18)
   END_RUNG
   // the same network as SCL:
   IF "On" AND "Timer".T30.Q AND NOT "DB08_Prestretch".dbx0_0 THEN "DB08_Prestretch".dbw20 := 202; END_IF;
   #_w1 := "On" AND "DB08_Prestretch".dbx0_0 AND NOT "Auto";
   IF #_w1 THEN "DB08_Prestretch".dbw20 := "DB26".Dbw88 + 100; END_IF;
   IF #_w1 AND ("DB26".Dbw88 <= 0) THEN "DB08_Prestretch".dbw20 := "DB26".Dbw88 + 101; END_IF;
   IF "On" AND "DB22_DisplayData".dbx15_1 THEN "DB08_Prestretch".dbw20 := 210; END_IF;
   IF "On" AND NOT "A15" THEN "DB08_Prestretch".dbw20 := 0; END_IF;
   IF "On" THEN "DB08_Prestretch".dbw18 := "DB08_Prestretch".dbw20; END_IF;
END_REGION

REGION Network 13
   RUNG wire#powerrail
      Contact( "On" )
      wire#w1
      Contact( "Auto" )
      { S7_GenerateENO := "TRUE" } Move(in := "DB03_Machine".dbw82, out1 => "DB08_Prestretch".dbw32)
   END_RUNG
   RUNG wire#w1
      Contact( "M1.1" )
      wire#w2
      { S7_GenerateENO := "TRUE" } Move(in := "DB250_ProgramData".Program.FilmPrestretchFinalRev, out1 => "DB08_Prestretch".dbw32)
   END_RUNG
   RUNG wire#w1
      Contact( "M1.2" )
   END_RUNG wire#w2
   RUNG wire#w1
      Contact( "M1.3" )
   END_RUNG wire#w2
   RUNG wire#w1
      Contact( "M1.4" )
   END_RUNG wire#w2
   RUNG wire#w1
      Contact( "ClampCutOk8" )
   END_RUNG wire#w2
   RUNG wire#w1
      Contact( "DB08_Prestretch".dbx0_0 )
      I_Contact( "Auto" )
      { S7_GenerateENO := "TRUE" } Move(in := "DB26".Dbw50, out1 => "DB08_Prestretch".dbw32)
   END_RUNG
   // the same network as SCL:
   IF "On" AND "Auto" THEN "DB08_Prestretch".dbw32 := "DB03_Machine".dbw82; END_IF;
   IF "On" AND ("M1.1" OR "M1.2" OR "M1.3" OR "M1.4" OR "ClampCutOk8") THEN
       "DB08_Prestretch".dbw32 := "DB250_ProgramData".Program.FilmPrestretchFinalRev;
   END_IF;
   IF "On" AND "DB08_Prestretch".dbx0_0 AND NOT "Auto" THEN "DB08_Prestretch".dbw32 := "DB26".Dbw50; END_IF;
END_REGION

REGION Network 14
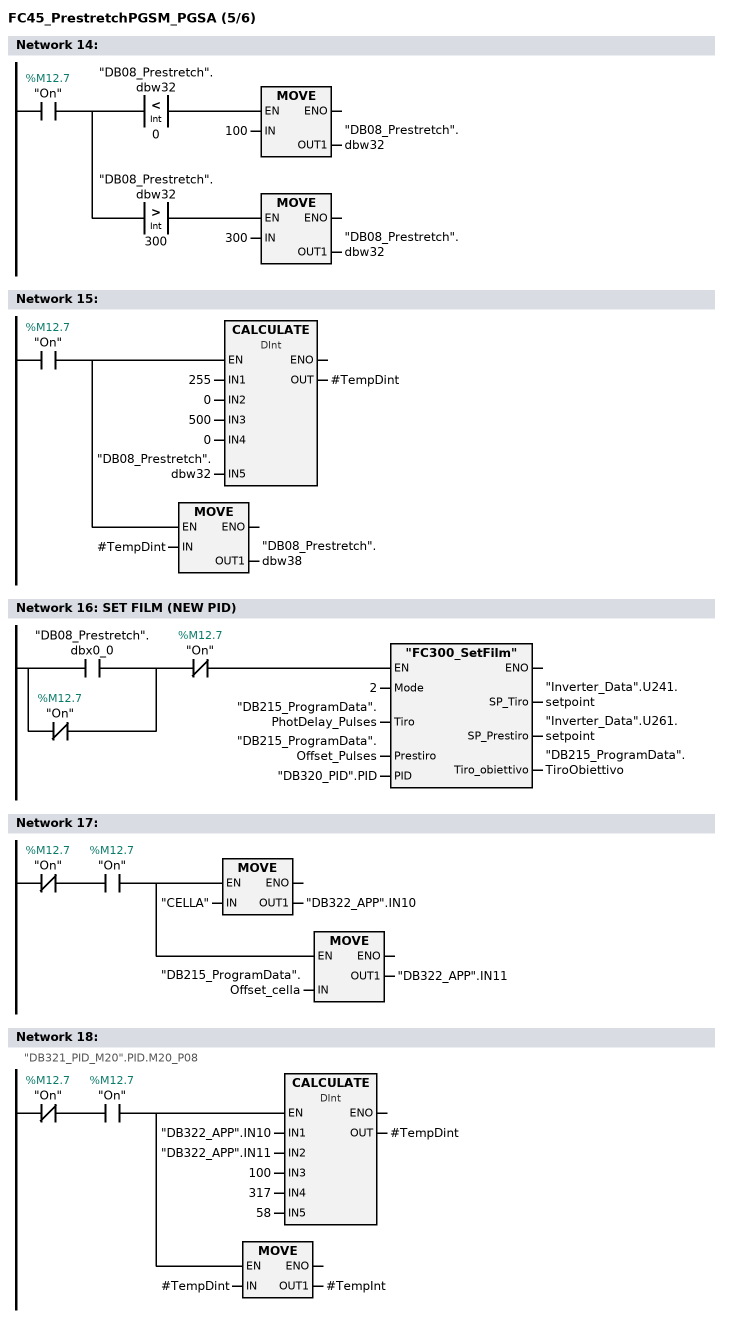
   RUNG wire#powerrail
      Contact( "On" )
      wire#w1
      { S7_Templates := "SrcType := Int" } LT_Contact(in1 := "DB08_Prestretch".dbw32, in2 := 0)
      { S7_GenerateENO := "TRUE" } Move(in := 100, out1 => "DB08_Prestretch".dbw32)
   END_RUNG
   RUNG wire#w1
      { S7_Templates := "SrcType := Int" } GT_Contact(in1 := "DB08_Prestretch".dbw32, in2 := 300)
      { S7_GenerateENO := "TRUE" } Move(in := 300, out1 => "DB08_Prestretch".dbw32)
   END_RUNG
   // the same network as SCL:
   IF "On" AND ("DB08_Prestretch".dbw32 < 0) THEN "DB08_Prestretch".dbw32 := 100; END_IF;
   IF "On" AND ("DB08_Prestretch".dbw32 > 300) THEN "DB08_Prestretch".dbw32 := 300; END_IF;
END_REGION

REGION Network 15
   RUNG wire#powerrail
      Contact( "On" )
      wire#w1
      { S7_Templates := "SrcType := DInt"; S7_GenerateENO := "TRUE"; S7_Expression := "((IN5-IN4)*(IN1-IN2)/(IN3-IN4))+IN2" } Calculate(in1 := 255, in2 := 0, in3 := 500, in4 := 0, in5 := "DB08_Prestretch".dbw32, out => #TempDint)
   END_RUNG
   RUNG wire#w1
      { S7_GenerateENO := "TRUE" } Move(in := #TempDint, out1 => "DB08_Prestretch".dbw38)
   END_RUNG
   // the same network as SCL:
   IF "On" THEN
       #TempDint := (("DB08_Prestretch".dbw32-0)*(255-0)/(500-0))+0;
       "DB08_Prestretch".dbw38 := #TempDint;
   END_IF;
END_REGION

REGION Network 16: SET FILM (NEW PID)
   RUNG wire#powerrail
      Contact( "DB08_Prestretch".dbx0_0 )
      wire#w1
      I_Contact( "On" )
      "FC300_SetFilm"(Mode := 2, Tiro := "DB215_ProgramData".PhotDelay_Pulses, Prestiro := "DB215_ProgramData".Offset_Pulses, PID := "DB320_PID".PID, SP_Tiro => "Inverter_Data".U241.setpoint, SP_Prestiro => "Inverter_Data".U261.setpoint, Tiro_obiettivo => "DB215_ProgramData".TiroObiettivo)
   END_RUNG
   RUNG wire#powerrail
      I_Contact( "On" )
   END_RUNG wire#w1
   // the same network as SCL:
   IF ("DB08_Prestretch".dbx0_0 OR NOT "On") AND NOT "On" THEN
       "FC300_SetFilm"(Mode := 2,
                       Tiro := "DB215_ProgramData".PhotDelay_Pulses,
                       Prestiro := "DB215_ProgramData".Offset_Pulses,
                       PID := "DB320_PID".PID,
                       SP_Tiro => "Inverter_Data".U241.setpoint,
                       SP_Prestiro => "Inverter_Data".U261.setpoint,
                       Tiro_obiettivo => "DB215_ProgramData".TiroObiettivo);
   END_IF;
END_REGION

REGION Network 17
   RUNG wire#powerrail
      I_Contact( "On" )
      Contact( "On" )
      wire#w1
      Move(in := "CELLA", out1 => "DB322_APP".IN10)
   END_RUNG
   RUNG wire#w1
      Move(in := "DB215_ProgramData".Offset_cella, out1 => "DB322_APP".IN11)
   END_RUNG
   // the same network as SCL:
   IF NOT "On" AND "On" THEN
       "DB322_APP".IN10 := "CELLA";
       "DB322_APP".IN11 := "DB215_ProgramData".Offset_cella;
   END_IF;
END_REGION

REGION Network 18
   // "DB321_PID_M20".PID.M20_P08
   RUNG wire#powerrail
      I_Contact( "On" )
      Contact( "On" )
      wire#w1
      { S7_Templates := "SrcType := DInt"; S7_Expression := "((IN1-IN2)*IN3/IN4)+IN5" } Calculate(in1 := "DB322_APP".IN10, in2 := "DB322_APP".IN11, in3 := 100, in4 := 317, in5 := 58, out => #TempDint)
   END_RUNG
   RUNG wire#w1
      Move(in := #TempDint, out1 => #TempInt)
   END_RUNG
   // the same network as SCL:
   IF NOT "On" AND "On" THEN
       #TempDint := (("DB322_APP".IN10-"DB322_APP".IN11)*100/317)+58;
       #TempInt := #TempDint;
   END_IF;
END_REGION

REGION Network 19
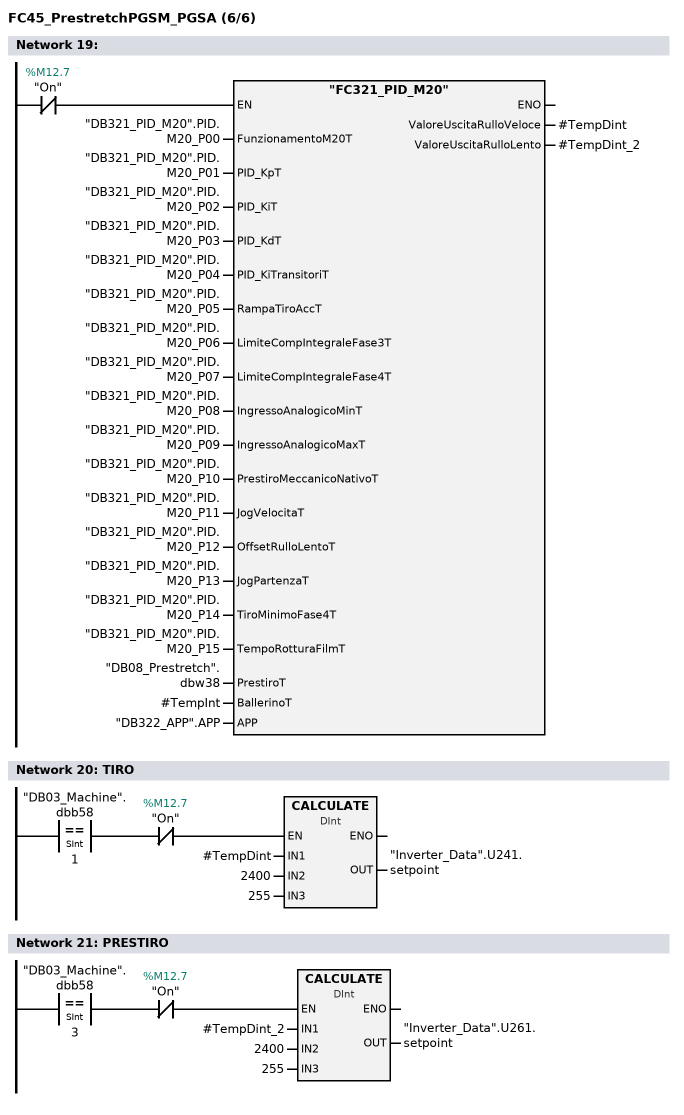
   RUNG wire#powerrail
      I_Contact( "On" )
      "FC321_PID_M20"(FunzionamentoM20T := "DB321_PID_M20".PID.M20_P00, PID_KpT := "DB321_PID_M20".PID.M20_P01, PID_KiT := "DB321_PID_M20".PID.M20_P02, PID_KdT := "DB321_PID_M20".PID.M20_P03, PID_KiTransitoriT := "DB321_PID_M20".PID.M20_P04, RampaTiroAccT := "DB321_PID_M20".PID.M20_P05, LimiteCompIntegraleFase3T := "DB321_PID_M20".PID.M20_P06, LimiteCompIntegraleFase4T := "DB321_PID_M20".PID.M20_P07, IngressoAnalogicoMinT := "DB321_PID_M20".PID.M20_P08, IngressoAnalogicoMaxT := "DB321_PID_M20".PID.M20_P09, PrestiroMeccanicoNativoT := "DB321_PID_M20".PID.M20_P10, JogVelocitaT := "DB321_PID_M20".PID.M20_P11, OffsetRulloLentoT := "DB321_PID_M20".PID.M20_P12, JogPartenzaT := "DB321_PID_M20".PID.M20_P13, TiroMinimoFase4T := "DB321_PID_M20".PID.M20_P14, TempoRotturaFilmT := "DB321_PID_M20".PID.M20_P15, PrestiroT := "DB08_Prestretch".dbw38, BallerinoT := #TempInt, APP := "DB322_APP".APP, ValoreUscitaRulloVeloce => #TempDint, ValoreUscitaRulloLento => #TempDint_2)
   END_RUNG
   // the same network as SCL:
   IF NOT "On" THEN
       "FC321_PID_M20"(FunzionamentoM20T := "DB321_PID_M20".PID.M20_P00,
                       PID_KpT := "DB321_PID_M20".PID.M20_P01,
                       PID_KiT := "DB321_PID_M20".PID.M20_P02,
                       PID_KdT := "DB321_PID_M20".PID.M20_P03,
                       PID_KiTransitoriT := "DB321_PID_M20".PID.M20_P04,
                       RampaTiroAccT := "DB321_PID_M20".PID.M20_P05,
                       LimiteCompIntegraleFase3T := "DB321_PID_M20".PID.M20_P06,
                       LimiteCompIntegraleFase4T := "DB321_PID_M20".PID.M20_P07,
                       IngressoAnalogicoMinT := "DB321_PID_M20".PID.M20_P08,
                       IngressoAnalogicoMaxT := "DB321_PID_M20".PID.M20_P09,
                       PrestiroMeccanicoNativoT := "DB321_PID_M20".PID.M20_P10,
                       JogVelocitaT := "DB321_PID_M20".PID.M20_P11,
                       OffsetRulloLentoT := "DB321_PID_M20".PID.M20_P12,
                       JogPartenzaT := "DB321_PID_M20".PID.M20_P13,
                       TiroMinimoFase4T := "DB321_PID_M20".PID.M20_P14,
                       TempoRotturaFilmT := "DB321_PID_M20".PID.M20_P15,
                       PrestiroT := "DB08_Prestretch".dbw38,
                       BallerinoT := #TempInt,
                       APP := "DB322_APP".APP,
                       ValoreUscitaRulloVeloce => #TempDint,
                       ValoreUscitaRulloLento => #TempDint_2);
   END_IF;
END_REGION

REGION Network 20: TIRO
   RUNG wire#powerrail
      { S7_Templates := "SrcType := SInt" } EQ_Contact(in1 := "DB03_Machine".dbb58, in2 := 1)
      I_Contact( "On" )
      { S7_Templates := "SrcType := DInt"; S7_Expression := "IN1*IN2/IN3" } Calculate(in1 := #TempDint, in2 := 2400, in3 := 255, out => "Inverter_Data".U241.setpoint)
   END_RUNG
   // the same network as SCL:
   IF ("DB03_Machine".dbb58 = 1) AND NOT "On" THEN
       "Inverter_Data".U241.setpoint := #TempDint*2400/255;
   END_IF;
END_REGION

REGION Network 21: PRESTIRO
   RUNG wire#powerrail
      { S7_Templates := "SrcType := SInt" } EQ_Contact(in1 := "DB03_Machine".dbb58, in2 := 3)
      I_Contact( "On" )
      { S7_Templates := "SrcType := DInt"; S7_Expression := "IN1*IN2/IN3" } Calculate(in1 := #TempDint_2, in2 := 2400, in3 := 255, out => "Inverter_Data".U261.setpoint)
   END_RUNG
   // the same network as SCL:
   IF ("DB03_Machine".dbb58 = 3) AND NOT "On" THEN
       "Inverter_Data".U261.setpoint := #TempDint_2*2400/255;
   END_IF;
END_REGION
END_FUNCTION

FUNCTION "FC300_SetFilm" : Void
{ S7_Optimized_Access := 'TRUE' }
VERSION : 0.1
   VAR_INPUT 
      Mode : UInt;
      Tiro : UInt;
      Prestiro : UInt;
   END_VAR

   VAR_OUTPUT 
      SP_Tiro : Real;
      SP_Prestiro : Real;
      Tiro_obiettivo : UInt;
   END_VAR

   VAR_IN_OUT 
      PID : "PID";
   END_VAR

   VAR_TEMP 
      freqT : DInt;
      freqP : DInt;
      tempo : UInt;
      t_temp : Time;
      velocita : DInt;
      correttivoTiro : UInt;
      correttivoPrestiro : UInt;
      rapporto : DInt;
      tiro_temp : UInt;
      clock : Bool;
   END_VAR

   VAR CONSTANT 
      BASE_PRESTIRO : UInt := 100;
      MAX_PRESTIRO_T0 : UInt := 75;
      MAX_PRESTIRO_PVS : UInt := 400;
      RAPP_PRES : UInt := 200;
   END_VAR


BEGIN
	(**)
	
	#freqT := 0;
	#freqP := 0;
	
	//Copia del valore di tiro per confronti in gestione RAMPA [partenza/fine ciclo] (OB30)
	#Tiro_obiettivo := #Tiro;
	
	IF (#PID.setTiro) THEN
	    //Fisso il tiro obiettivo senza passare dalla rampa. Mi serve in avvio ciclo o quando riparto
	    //#PID.tiro := #Tiro;
	    #PID.setTiro := FALSE;
	    //"SetFilmStep" := 1;
	END_IF;
	
	//#tiro_temp := #PID.tiro;
	
	//CARRELLO PVS
	//
	IF (#Mode = 2) THEN //FILM_RUN
	    //Eseguo il calcolo dei parametri (PID) solo ad ogni nuovo valore letto dalla cella (scheda prestiro)
	    IF ("PrestNewValue") THEN
	        "FC320_PID_ParamCalc"(Tiro := #PID.tiro,
	                              Offset_cella := "DB215_ProgramData".Offset_cella,
	                              PID := #PID);
	        "PrestNewValue" := 0;
	    END_IF;
	    //Frequenza TIRO
	    #velocita := #PID.segnale;
	    #freqT := #velocita;
	    (*
	    //Correttivo TIRO
	    #correttivoTiro := (#MAX_PRESTIRO_T0 - 15);//"DB230_Parameters".P_PRESTMIN);
	    #correttivoTiro := (#correttivoTiro * (100 - #Tiro)) / 100;
	    //CorrettivoPRESTIRO
	    #correttivoPrestiro := ((#MAX_PRESTIRO_PVS - #Prestiro) * #Tiro) / 500;
	    //    
	    #rapporto := #BASE_PRESTIRO + #correttivoTiro - #correttivoPrestiro;
	    #rapporto := #rapporto + #Prestiro;
	    #rapporto := #rapporto + 15;//"DB230_Parameters".P_PRESTMIN;
	    //    
	    #velocita := #velocita * #RAPP_PRES;
	    #velocita := #velocita / #rapporto;
	    *)
	    //Frequenza PRESTIRO
	    #rapporto := #BASE_PRESTIRO + #Prestiro;
	    #freqP := #velocita * #RAPP_PRES / #rapporto;
	    //#freqP := #velocita*2/5;
	    //
	    //SP_INVERTER SIEMENS IN RPM (1500@50HZ) -> CONVERSIONE SECONDO PROPORZIONE    
	    #SP_Tiro := DINT_TO_REAL(#freqT * 5);//10);//10);
	    IF (#SP_Tiro >= 3000.0) THEN
	        #SP_Tiro := 3000.0;
	    END_IF;
	    #SP_Prestiro := DINT_TO_REAL(#freqP * 5);//10);//10);
	    IF (#SP_Prestiro >= 3000.0) THEN
	        #SP_Prestiro := 3000.0;
	    END_IF;
	    //
	ELSIF (#Mode = 1) THEN  // FILM_STOP - Freq.Rulli = 0 (per strappare il film durante il taglio)
	    #SP_Tiro := 0;
	    #SP_Prestiro := 0;
	ELSIF (#Mode = 3) THEN     // FILM_MANUAL - Svolgimento film in manuale
	    #SP_Tiro := 1500;
	    #SP_Prestiro := 1500;
	ELSIF (#Mode = 0) THEN    // FILM_DISABLE
	    #SP_Tiro := 0;
	    #SP_Prestiro := 0;
	END_IF;
	//
	(*
	//Film rotto o esaurito
	//
	//IF "CELLA" >= ("DB215_ProgramData".Offset_cella + 10) AND "Timer".T21.Q THEN
	//
	IF "DB230_Parameters".FilmEndEn THEN
	    IF "DB02_Timers".T021.Q THEN
	        "FilmEnd" := 1;
	        "FilmEnd2" := 1;
	    END_IF;
	    IF "DB200_Supervisor".State_Stop = 110 THEN
	        "FilmEnd" := 0;
	    END_IF;
	END_IF;
	*)
END_FUNCTION

FUNCTION "FC321_PID_M20" : Void
{ S7_Optimized_Access := 'TRUE' }
VERSION : 0.1
   VAR_INPUT 
      FunzionamentoM20T : Int;
      PID_KpT : Int;
      PID_KiT : Int;
      PID_KdT : Int;
      PID_KiTransitoriT : Int;
      RampaTiroAccT : Int;
      LimiteCompIntegraleFase3T : Int;
      LimiteCompIntegraleFase4T : Int;
      IngressoAnalogicoMinT : Int;
      IngressoAnalogicoMaxT : Int;
      PrestiroMeccanicoNativoT : Int;
      JogVelocitaT : Int;
      OffsetRulloLentoT : Int;
      JogPartenzaT : Int;
      TiroMinimoFase4T : Int;
      TempoRotturaFilmT : Int;
      PrestiroT : Int;
      BallerinoT : Int;
   END_VAR

   VAR_OUTPUT 
      ValoreUscitaRulloVeloce : DInt;
      ValoreUscitaRulloLento : DInt;
   END_VAR

   VAR_IN_OUT 
      APP : "APP";
   END_VAR

   VAR_TEMP 
      PID_ComponenteProporzionale : DInt;
      PID_ComponenteIntegrale : DInt;
      PID_ComponenteDerivativa : DInt;
      Tiro : Int;
      Tiro1 : Int;
      Tiro2 : Int;
      TiroPrecedente : Int;
      TiroAppoggio : Int;
      ErroreAttuale : Int;
      ErrorePrecedente : Int;
      PID_Kp : Int;
      PID_Ki : Int;
      PID_Kd : Int;
      SetpointTiro : Int;
      SetpointTiroRampa : Int;
      TransitorioInizialeFase1 : Int;
      TransitorioFase3 : Int;
      TransitorioFase4 : Int;
      VelocitaRotazione : Int;
      VelocitaRotazioneFase2 : Int;
      VelocitaRotazioneAppoggio1 : Int;
      VelocitaRotazioneAppoggio2 : Int;
      Fase1OneShoot : Int;
      Fase2OneShoot : Int;
      Fase3OneShoot : Int;
      Fase4OneShoot : Int;
      ArrestoRepentinoOneShoot : Int;
      TiroFase1 : Int;
      TempIntero : Int;
      Fase : Int;
      BallerinoPrecedente : Array[0..2] of Int;
      LimiteComponenteIntegrale : Int;
      TiroRichiesto : Int;
      TimerArrestoRepentino : Int;
      TiroMinimoArrestoRepentino : Int;
      VariazioneTiro : Int;
      TimerFase2 : Int;
      TempoRotturaFilm : Int;
      TimerFase4 : Int;
      TiroMinimoFase4 : Int;
      PID_Uscita : DInt;
      PrestiroRichiesto : DInt;
      PrestiroAppoggio : Real;
   END_VAR

   VAR CONSTANT 
      PID_LimiteSuperioreIntegrale : DInt := 23000;
      PID_LimiteInferioreIntegrale : DInt := 0;
      PID_LimiteSuperioreDerivativa : DInt := 6000;
      PID_LimiteInferioreDerivativa : DInt := -6000;
      PID_LimiteSuperioreUscita : DInt := 255;
      PID_LimiteInferioreUscita : DInt := 0;
   END_VAR


BEGIN
	// Devono esserci due letture uguali per cambiare il valore di tiro. Serve a filtrare letture spurie
	//
	#APP.Tiro1 := "DB08_Prestretch".dbw18; //val_parametro[22];
	//
	IF (#APP.Tiro1 = #APP.Tiro2) THEN
	    #APP.Tiro := #APP.#Tiro1;
	END_IF;
	//
	#APP.Tiro2 := #APP.#Tiro1;
	//
	#APP.VelocitaRotazione := "DB09_TablePos".dbw10; //val_parametro[20];
	//
	// Fase 1:  Accelerazione
	//***********************
	IF (#APP.Tiro = 206) THEN
	    #APP.Fase := 1;
	    //Inizializzazione Fase 1
	    IF (#APP.Fase1OneShoot = 0) THEN
	        #APP.SetpointTiroRampa := #BallerinoT * 10;
	        #APP.TransitorioInizialeFase1 := 1;
	        #APP.Fase1OneShoot := 1;
	        #APP.PID_ComponenteIntegrale := #APP.PID_ComponenteIntegrale + #JogPartenzaT * 100; //Incremento di componente integrale per limitare tiri alti alla partenza 
	    END_IF;
	    //
	    #APP.VariazioneTiro := #BallerinoT - #APP.BallerinoPrecedente[2];
	    //#APP.VariazioneTiro := (#BallerinoT - #APP.BallPrec_2);
	    #APP.PID_Kp := #PID_KpT * 2;
	    #APP.PID_Ki := #PID_KiT * 2;
	    #APP.PID_Kd := #PID_KdT * 3;
	    //
	    IF (#APP.VariazioneTiro < 0) THEN
	        #APP.PID_Kd := 0;
	    END_IF;
	    //
	    IF (#APP.TiroFase1 = 0) THEN
	        #APP.TiroFase1 := 5;
	    END_IF;
	    //
	    #APP.SetpointTiro := ((#IngressoAnalogicoMaxT - #IngressoAnalogicoMinT) * #APP.TiroFase1 / 100) + #IngressoAnalogicoMinT;
	    //
	    //Incremento componente integrale durante la fase di accelerazione per ridurre l'errore sul tiro desiderato
	    IF (#APP.VariazioneTiro > 0 AND #APP.ErroreAttuale > 0) THEN
	        IF (#FunzionamentoM20T = 0) THEN
	            #APP.PID_ComponenteIntegrale := #APP.PID_ComponenteIntegrale + #PID_KpT * #APP.ErroreAttuale / 4;
	        ELSE //(#APP.FunzionamentoM20T == 1)
	            #APP.PID_ComponenteIntegrale := #APP.PID_ComponenteIntegrale + #PID_KpT * #APP.ErroreAttuale / 10;
	        END_IF;
	    END_IF;
	    //Rampa di tiro per tiri alti
	    IF (#APP.TransitorioInizialeFase1 = 1) THEN
	        IF (#APP.SetpointTiroRampa / 10 < #APP.SetpointTiro) THEN
	            #APP.SetpointTiroRampa := #APP.SetpointTiroRampa + #RampaTiroAccT;
	            #APP.SetpointTiro := #APP.SetpointTiroRampa / 10;
	        ELSE
	            #APP.TransitorioInizialeFase1 := 0;
	        END_IF;
	    END_IF;
	    #APP.TiroRichiesto := #APP.TiroFase1;
	END_IF;
	//
	// Fase 2: Fasciatura a regime
	//****************************
	IF (#APP.Tiro > 0 AND #APP.Tiro <= 100) THEN
	    #APP.Fase := 2;
	    #APP.Fase4OneShoot := 0;
	    // Inizializzazione Fase 2      
	    IF (#APP.Fase2OneShoot = 0) THEN
	        #APP.VelocitaRotazioneFase2 := 0;
	        #APP.Fase2OneShoot := 1;
	        // PID_ComponenteIntegrale = PID_ComponenteIntegrale+2000; //Fornisco un piccolo delta di velocita'alla partenza per evitare di tirare strattoni sul ballerino all'avvio 
	    END_IF;
	    #APP.PID_Kp := #PID_KpT;
	    #APP.PID_Ki := #PID_KiT;
	    #APP.PID_Kd := #PID_KdT;
	    IF (#APP.Tiro >= 50) THEN
	        #APP.PID_Ki := (15 + 20 * #PID_KiT) / 30; //Per tiri alti diminuisco il guadagno integrale per rendere il regolatore meno pronto e farlo oscillare meno.
	    END_IF;
	    #APP.SetpointTiro := ((#IngressoAnalogicoMaxT - #IngressoAnalogicoMinT) * #APP.Tiro / 100) + #IngressoAnalogicoMinT;
	    #APP.TiroFase1 := #APP.Tiro;
	    //
	    //Velocita' di rotazione braccio nella Fase 2. Filtro di 3 scansioni
	    IF (#APP.VelocitaRotazione = #APP.VelocitaRotazioneAppoggio1 AND #APP.VelocitaRotazioneAppoggio1 = #APP.VelocitaRotazioneAppoggio2) THEN
	        #APP.VelocitaRotazioneFase2 := #APP.VelocitaRotazione;
	    END_IF;
	    #APP.VelocitaRotazioneAppoggio2 := #APP.VelocitaRotazioneAppoggio1;
	    #APP.VelocitaRotazioneAppoggio1 := #APP.VelocitaRotazione;
	    //
	    //Rottura film
	    IF (#BallerinoT < #IngressoAnalogicoMinT) THEN
	        #APP.TimerFase2 := #APP.TimerFase2 + 1;
	    ELSE
	        #APP.TimerFase2 := 0;
	    END_IF;
	    //
	    #APP.TempoRotturaFilm := #TempoRotturaFilmT * 10 / 3; //Tempo rottura film in numero di scansioni
	    IF (#APP.TimerFase2 >= #APP.TempoRotturaFilm) THEN
	        #APP.PID_ComponenteIntegrale := 0;
	        #APP.TimerFase2 := 0;
	    END_IF;
	    #APP.TiroRichiesto := #APP.Tiro;
	END_IF;
	//
	// Fase 3: Transitorio velocita' alta -> media
	//********************************************
	IF (#APP.Tiro > 100 AND #APP.Tiro <= 200) THEN
	    #APP.Fase := 3;
	    #APP.Fase4OneShoot := 0;
	    //
	    // Inizializzazione Fase 3
	    IF (#APP.Fase3OneShoot = 0) THEN
	        #APP.TransitorioFase3 := 0;
	        #APP.Fase3OneShoot := 1;
	    END_IF;
	    //
	    #APP.LimiteComponenteIntegrale := #LimiteCompIntegraleFase3T * 100;
	    #APP.PID_Kp := #PID_KpT;
	    #APP.PID_Ki := #PID_KiTransitoriT;
	    #APP.PID_Kd := #PID_KdT;
	    #APP.SetpointTiro := ((#IngressoAnalogicoMaxT - #IngressoAnalogicoMinT) * (#APP.Tiro - 100) / 100) + #IngressoAnalogicoMinT;
	    //
	    #APP.TempIntero := #APP.VelocitaRotazioneFase2 * 9 / 10;
	    IF (#APP.VelocitaRotazione < #APP.TempIntero AND #APP.TransitorioFase3 = 0) THEN
	        #APP.TransitorioFase3 := 1;
	        IF (#APP.PID_ComponenteIntegrale > #APP.LimiteComponenteIntegrale) THEN
	            #APP.PID_ComponenteIntegrale := #APP.LimiteComponenteIntegrale;
	        END_IF;
	    END_IF;
	    #APP.TiroRichiesto := #APP.Tiro - 100;
	END_IF;
	//
	// Fase 4: Transitorio velocita' media -> bassa
	// ********************************************
	IF (#APP.Tiro = 201) THEN
	    #APP.Fase := 4;
	    // Inizializzazione Fase 4
	    IF (#APP.Fase4OneShoot = 0) THEN
	        #APP.TransitorioFase4 := 0;
	        #APP.Fase4OneShoot := 1;
	    END_IF;
	    //
	    IF (#APP.TiroPrecedente <= 100) THEN
	        #APP.TiroAppoggio := #APP.TiroPrecedente;
	    END_IF;
	    //
	    IF (#APP.TiroPrecedente > 100 AND #APP.TiroPrecedente <= 200) THEN
	        #APP.TiroAppoggio := #APP.TiroPrecedente - 100;
	    END_IF;
	    //
	    //Alzo il tiro richiesto nei primi decimi, in maniera da abbattere la componente integrale
	    #APP.TiroMinimoFase4 := #TiroMinimoFase4T;
	    //
	    IF (#APP.TiroAppoggio < #APP.TiroMinimoFase4) THEN
	        #APP.TiroAppoggio := #APP.TiroMinimoFase4;
	    END_IF;
	    //
	    #APP.SetpointTiro := ((#IngressoAnalogicoMaxT - #IngressoAnalogicoMinT) * #APP.TiroAppoggio / 100) + #IngressoAnalogicoMinT;
	    //
	    #APP.LimiteComponenteIntegrale := #LimiteCompIntegraleFase4T * 100;
	    #APP.PID_Kp := #PID_KpT;
	    #APP.PID_Ki := #PID_KiTransitoriT * 15 / 10;
	    #APP.PID_Kd := #PID_KdT;
	    IF (#APP.PID_ComponenteIntegrale > #APP.LimiteComponenteIntegrale) THEN
	        #APP.PID_ComponenteIntegrale := #APP.LimiteComponenteIntegrale;
	    END_IF;
	    //
	    #APP.TransitorioFase4 := 1;
	    #APP.TiroRichiesto := #APP.TiroAppoggio;
	END_IF;
	//
	// Fase 0: Azzeramento del regolatore
	// **********************************
	IF (#APP.Tiro = 0) THEN
	    #APP.Fase := 0;
	    #APP.PID_ComponenteIntegrale := 0;
	    #APP.Fase1OneShoot := 0;
	    #APP.Fase2OneShoot := 0;
	    #APP.Fase3OneShoot := 0;
	    #APP.Fase4OneShoot := 0;
	    #APP.ArrestoRepentinoOneShoot := 0;
	    #APP.SetpointTiro := #BallerinoT;
	    #APP.TiroPrecedente := 0;
	    #APP.TiroFase1 := 0;
	    #APP.TiroAppoggio := 0;
	END_IF;
	//   
	// Jog in manuale
	// **************
	IF (#APP.Tiro = 210) THEN
	    #APP.PID_Kp := 0;
	    #APP.PID_Ki := 0;
	    #APP.PID_Kd := 0;
	    #APP.PID_ComponenteIntegrale := #JogVelocitaT * 100;
	END_IF;
	//   
	// Arresto repentino
	// *****************
	IF (#APP.Tiro = 202) THEN
	    // Inizializzazione Fase 4
	    IF (#APP.ArrestoRepentinoOneShoot = 0) THEN
	        #APP.TimerArrestoRepentino := 0;
	        #APP.ArrestoRepentinoOneShoot := 1;
	    END_IF;
	    //
	    #APP.TimerArrestoRepentino := #APP.TimerArrestoRepentino + 1;
	    #APP.TiroMinimoArrestoRepentino := #TiroMinimoFase4T * 175 / 100;
	    //
	    IF (#APP.TiroPrecedente <= 100) THEN
	        #APP.TiroAppoggio := #APP.TiroPrecedente;
	    END_IF;
	    //
	    IF (#APP.TiroPrecedente > 100 & #APP.TiroPrecedente <= 200) THEN
	        #APP.TiroAppoggio := #APP.TiroPrecedente - 100;
	    END_IF;
	    //
	    IF (#APP.TiroAppoggio < #APP.TiroMinimoArrestoRepentino) THEN
	        #APP.TiroAppoggio := #APP.TiroMinimoArrestoRepentino;
	    END_IF;
	    //
	    #APP.SetpointTiro := ((#IngressoAnalogicoMaxT - #IngressoAnalogicoMinT) * #APP.TiroAppoggio / 100) + #IngressoAnalogicoMinT;
	    //   
	    #APP.PID_Kp := #PID_KpT;
	    #APP.PID_Ki := #PID_KiTransitoriT * 175 / 100;
	    #APP.PID_Kd := #PID_KdT;
	    //
	    #APP.TiroRichiesto := #APP.TiroAppoggio;
	END_IF;
	//
	// Regolatore PID standard 
	#APP.ErroreAttuale := (#BallerinoT - #APP.SetpointTiro);
	//
	// Componente proporzionale del regolatore          
	#APP.PID_ComponenteProporzionale := #APP.PID_Kp * #APP.ErroreAttuale;
	//
	// Componente integrale del regolatore
	#APP.PID_ComponenteIntegrale := #APP.PID_ComponenteIntegrale + #APP.PID_Ki * #APP.ErroreAttuale / 10;
	//
	IF (#APP.PID_ComponenteIntegrale > #PID_LimiteSuperioreIntegrale AND #APP.Tiro <> 210) THEN
	    #APP.PID_ComponenteIntegrale := #PID_LimiteSuperioreIntegrale;
	END_IF;
	//
	IF (#APP.PID_ComponenteIntegrale > 25500 AND #APP.Tiro = 210) THEN
	    #APP.PID_ComponenteIntegrale := 25500;
	END_IF;
	//
	IF (#APP.PID_ComponenteIntegrale < #PID_LimiteInferioreIntegrale) THEN
	    #APP.PID_ComponenteIntegrale := #PID_LimiteInferioreIntegrale;
	END_IF;
	//
	// Componente derivativa del regolatore
	// PID_ComponenteDerivativa = 10*PID_Kd*(ErroreAttuale-ErrorePrecedente);
	
	#APP.PID_ComponenteDerivativa := 10 * #APP.PID_Kd * (#BallerinoT - #APP.BallerinoPrecedente[2]);
	
	//#PID_ComponenteDerivativa := 10 * #PID_Kd * (#BallerinoT - #APP.BallPrec_2);
	//
	IF (#APP.PID_ComponenteDerivativa > #PID_LimiteSuperioreDerivativa) THEN
	    #APP.PID_ComponenteDerivativa := #PID_LimiteSuperioreDerivativa;
	END_IF;
	//
	IF (#APP.PID_ComponenteDerivativa < #PID_LimiteInferioreDerivativa) THEN
	    #APP.PID_ComponenteDerivativa := #PID_LimiteInferioreDerivativa;
	END_IF;
	//
	#APP.PID_Uscita := (#APP.PID_ComponenteProporzionale + #APP.PID_ComponenteIntegrale + #APP.PID_ComponenteDerivativa) / 100; //Le costanti Kp, Ki e Kd sono espresse nel display in centesimi
	//
	IF (#APP.PID_Uscita > #PID_LimiteSuperioreUscita) THEN
	    #APP.PID_Uscita := #PID_LimiteSuperioreUscita;
	END_IF;
	//
	IF (#APP.PID_Uscita < #PID_LimiteInferioreUscita) THEN
	    #APP.PID_Uscita := #PID_LimiteInferioreUscita;
	END_IF;
	//
	IF (#APP.Tiro = 0) THEN
	    #APP.PID_Uscita := 0;
	END_IF;
	//
	// Aggiornamento valori precedenti  
	#APP.ErrorePrecedente := #APP.ErroreAttuale;
	//
	IF (#APP.Tiro <= 200) THEN
	    #APP.TiroPrecedente := #APP.Tiro;
	END_IF;
	//
	#APP.BallerinoPrecedente[2] := #APP.BallerinoPrecedente[1];
	#APP.BallerinoPrecedente[1] := #APP.BallerinoPrecedente[0];
	#APP.BallerinoPrecedente[0] := #BallerinoT;
	// #APP.BallPrec_2 := #APP.BallPrec_1;
	// #APP.BallPrec_1 := #APP.BallPrec_0;
	// #APP.BallPrec_0 := #BallerinoT;
	//
	// Attuazione delle uscite analogiche che vanno agli inverter
	#ValoreUscitaRulloVeloce := #APP.PID_Uscita;
	
	// Prestiro per PGSM e PGSA
	IF (#FunzionamentoM20T = 0) THEN
	    //
	    #APP.PrestiroRichiesto := INT_TO_DINT(#PrestiroT) * 500 / 255 + 100;
	    // Arrotonda sempre all'intero inferiore, a prescindere. Sommando 0.5 arrotondo all'intero piu vicino
	    #APP.PrestiroAppoggio := 0.5 + DINT_TO_REAL(#ValoreUscitaRulloVeloce * (#PrestiroMeccanicoNativoT + 100) / #APP.PrestiroRichiesto);
	    #APP.PrestiroAppoggio := #APP.PrestiroAppoggio + (#OffsetRulloLentoT - 10);
	    IF (#APP.PrestiroAppoggio > 255) THEN
	        #APP.PrestiroAppoggio := 255;
	    END_IF;
	    #ValoreUscitaRulloLento := REAL_TO_DINT(#APP.PrestiroAppoggio);
	END_IF;
	//
	// Tiro ballerino SCSP valvola proporzionale        
	IF (#FunzionamentoM20T = 1) THEN
	    #ValoreUscitaRulloLento := #PrestiroT;
	    IF (#ValoreUscitaRulloLento > 255) THEN
	        #ValoreUscitaRulloLento := 255;
	    END_IF;
	END_IF;
	
	
	
END_FUNCTION

FUNCTION "Inverter_CW_Assembly" : Void   // FC16, FBD
{ S7_Optimized_Access := 'TRUE' }
VERSION : 0.1
// stored: AutoNumber false, IsIECCheckEnabled false, SetENOAutomatically false, UDAEnableTagReadback false
   VAR_INPUT
      CW_Off1_On : Bool;
      CW_Off2 : Bool;
      CW_Off3 : Bool;
      CW_enable_operation : Bool;
      CW_no_lock_RFG : Bool;
      CW_no_stop_RFG : Bool;
      CW_enable_setpoint : Bool;
      CW_acknowledge : Bool;
      CW_not_used_1 : Bool;
      CW_not_used_2 : Bool;
      CW_PLC_is_Master : Bool;
      CW_direction_reversal : Bool;
      CW_not_used_3 : Bool;
      CW_motortpoti_up : Bool;
      CW_motortpoti_down : Bool;
      CW_not_used_4 : Bool;
   END_VAR
   VAR_IN_OUT
      Control_word : Word;
   END_VAR
BEGIN

REGION Network 1
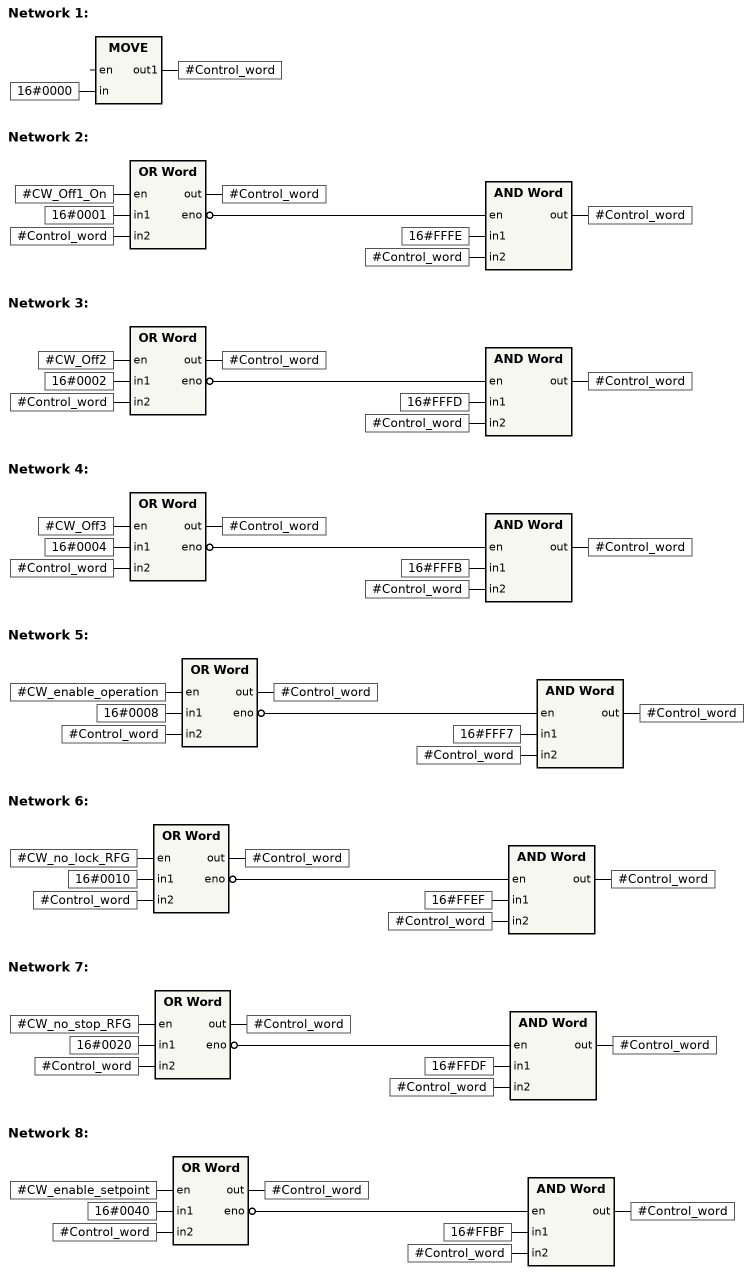
   #Control_word := 16#0000;
END_REGION

REGION Network 2
   IF #CW_Off1_On THEN #Control_word := 16#0001 OR #Control_word; END_IF;
   IF NOT #CW_Off1_On THEN #Control_word := 16#FFFE AND #Control_word; END_IF;
END_REGION

REGION Network 3
   IF #CW_Off2 THEN #Control_word := 16#0002 OR #Control_word; END_IF;
   IF NOT #CW_Off2 THEN #Control_word := 16#FFFD AND #Control_word; END_IF;
END_REGION

REGION Network 4
   IF #CW_Off3 THEN #Control_word := 16#0004 OR #Control_word; END_IF;
   IF NOT #CW_Off3 THEN #Control_word := 16#FFFB AND #Control_word; END_IF;
END_REGION

REGION Network 5
   IF #CW_enable_operation THEN #Control_word := 16#0008 OR #Control_word; END_IF;
   IF NOT #CW_enable_operation THEN #Control_word := 16#FFF7 AND #Control_word; END_IF;
END_REGION

REGION Network 6
   IF #CW_no_lock_RFG THEN #Control_word := 16#0010 OR #Control_word; END_IF;
   IF NOT #CW_no_lock_RFG THEN #Control_word := 16#FFEF AND #Control_word; END_IF;
END_REGION

REGION Network 7
   IF #CW_no_stop_RFG THEN #Control_word := 16#0020 OR #Control_word; END_IF;
   IF NOT #CW_no_stop_RFG THEN #Control_word := 16#FFDF AND #Control_word; END_IF;
END_REGION

REGION Network 8
   IF #CW_enable_setpoint THEN #Control_word := 16#0040 OR #Control_word; END_IF;
   IF NOT #CW_enable_setpoint THEN #Control_word := 16#FFBF AND #Control_word; END_IF;
END_REGION

REGION Network 9
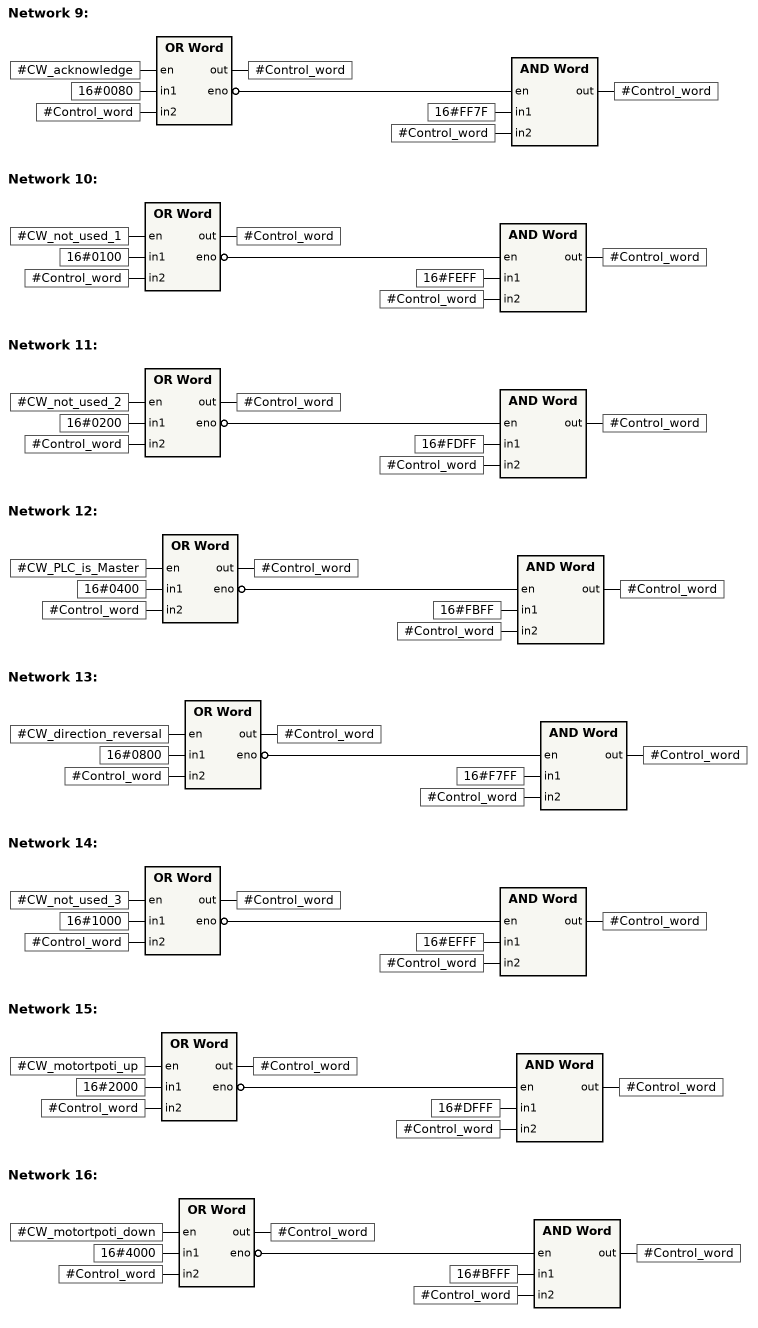
   IF #CW_acknowledge THEN #Control_word := 16#0080 OR #Control_word; END_IF;
   IF NOT #CW_acknowledge THEN #Control_word := 16#FF7F AND #Control_word; END_IF;
END_REGION

REGION Network 10
   IF #CW_not_used_1 THEN #Control_word := 16#0100 OR #Control_word; END_IF;
   IF NOT #CW_not_used_1 THEN #Control_word := 16#FEFF AND #Control_word; END_IF;
END_REGION

REGION Network 11
   IF #CW_not_used_2 THEN #Control_word := 16#0200 OR #Control_word; END_IF;
   IF NOT #CW_not_used_2 THEN #Control_word := 16#FDFF AND #Control_word; END_IF;
END_REGION

REGION Network 12
   IF #CW_PLC_is_Master THEN #Control_word := 16#0400 OR #Control_word; END_IF;
   IF NOT #CW_PLC_is_Master THEN #Control_word := 16#FBFF AND #Control_word; END_IF;
END_REGION

REGION Network 13
   IF #CW_direction_reversal THEN #Control_word := 16#0800 OR #Control_word; END_IF;
   IF NOT #CW_direction_reversal THEN #Control_word := 16#F7FF AND #Control_word; END_IF;
END_REGION

REGION Network 14
   IF #CW_not_used_3 THEN #Control_word := 16#1000 OR #Control_word; END_IF;
   IF NOT #CW_not_used_3 THEN #Control_word := 16#EFFF AND #Control_word; END_IF;
END_REGION

REGION Network 15
   IF #CW_motortpoti_up THEN #Control_word := 16#2000 OR #Control_word; END_IF;
   IF NOT #CW_motortpoti_up THEN #Control_word := 16#DFFF AND #Control_word; END_IF;
END_REGION

REGION Network 16
   IF #CW_motortpoti_down THEN #Control_word := 16#4000 OR #Control_word; END_IF;
   IF NOT #CW_motortpoti_down THEN #Control_word := 16#BFFF AND #Control_word; END_IF;
END_REGION

REGION Network 17
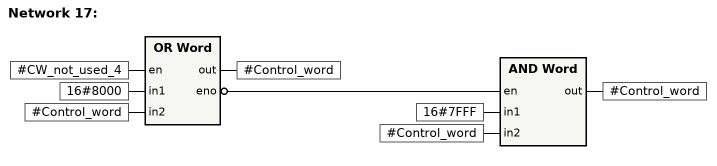
   IF #CW_not_used_4 THEN #Control_word := 16#8000 OR #Control_word; END_IF;
   IF NOT #CW_not_used_4 THEN #Control_word := 16#7FFF AND #Control_word; END_IF;
END_REGION
END_FUNCTION

FUNCTION_BLOCK "Inverter_Process_Data"   // FB1, FBD
{ S7_Optimized_Access := 'TRUE' }
VERSION : 0.1
// stored: AutoNumber false, IsIECCheckEnabled false, IsRetainMemResEnabled false, MemoryReserve 100, SetENOAutomatically false, UDAEnableTagReadback false
   VAR_INPUT
      control_word : Word := 16#0000;
      setpoint : Real;
      RD_address : HW_SUBMODULE;
      WR_address : HW_SUBMODULE;
      ref_quantity : Struct
         speed_p2000 : Real := 1500.0;
         current_p2002 : Real := 0.65;
         torque_p2003 : Real := 1.7;
      END_STRUCT;
   END_VAR
   VAR_OUTPUT
      status_word : Word;
      actual_speed : Real;
      actual_current : Real;
      actual_torque : Real;
      actual_alarm : Word;
      actual_fault : Word;
      RETVAL_RD : Word;
      RETVAL_WR : Word;
   END_VAR
   VAR_TEMP
      InData : Array[1..6] of Word;
      OutData : Array[1..6] of Word;
      actual_speed_INT : Int;
      actual_current_INT : Int;
      actual_torque_INT : Int;
      setpoint_INT : Int;
   END_VAR
BEGIN

REGION Network 1
